LIN {X 0,Y 518.239,Z 318.605,A -85,B 0,C 180,E1 -4964.129,E2 -4964.129} C_VEL
LIN {X 0,Y 518.643,Z 306.673,A -85,B 0,C 180,E1 -4964.92,E2 -4964.92} C_VEL
LIN {X 0,Y 519.008,Z 293.496,A -85,B 0,C 180,E1 -4965.613,E2 -4965.613} C_VEL
LIN {X 0,Y 519.32,Z 279.565,A -85,B 0,C 180,E1 -4966.165,E2 -4966.165} C_VEL
LIN {X 0,Y 519.404,Z 270.973,A -85,B 0,C 180,E1 -4966.425,E2 -4966.425} C_VEL
LIN {X 0,Y 516.398,Z 257.452,A -85,B 0,C 180,E1 -4966.836,E2 -4966.836} C_VEL
LIN {X 0,Y 516.463,Z 251.755,A -85,B 0,C 180,E1 -4970.124,E2 -4970.124} C_VEL
LIN {X 0,Y 516.525,Z 246.395,A -85,B 0,C 180,E1 -4973.24,E2 -4973.24} C_VEL
LIN {X 0,Y 516.572,Z 241.654,A -85,B 0,C 180,E1 -4976.112,E2 -4976.112} C_VEL
LIN {X 0,Y 516.692,Z 236.476,A -85,B 0,C 180,E1 -4979.319,E2 -4979.319} C_VEL
LIN {X 0,Y 516.772,Z 231.444,A -85,B 0,C 180,E1 -4982.521,E2 -4982.521} C_VEL
LIN {X 0,Y 516.881,Z 227.139,A -85,B 0,C 180,E1 -4985.332,E2 -4985.332} C_VEL
LIN {X 0,Y 516.903,Z 223.246,A -85,B 0,C 180,E1 -4987.946,E2 -4987.946} C_VEL
LIN {X 0,Y 516.84,Z 221.733,A -85,B 0,C 180,E1 -4989.187,E2 -4989.187} C_VEL
LIN {X 0,Y 516.914,Z 221.722,A -85,B 0,C 180,E1 -4991.775,E2 -4991.775} C_VEL
LIN {X 0,Y 516.926,Z 221.721,A -85,B 0,C 180,E1 -4995.01,E2 -4995.01} C_VEL
LIN {X 0,Y 516.895,Z 221.723,A -85,B 0,C 180,E1 -4998.402,E2 -4998.402} C_VEL
LIN {X 0,Y 516.879,Z 221.728,A -85,B 0,C 180,E1 -5001.284,E2 -5001.284} C_VEL
LIN {X 0,Y 516.874,Z 221.728,A -85,B 0,C 180,E1 -5004.22,E2 -5004.22} C_VEL
LIN {X 0,Y 516.884,Z 221.723,A -85,B 0,C 180,E1 -5007.052,E2 -5007.052} C_VEL
LIN {X 0,Y 516.872,Z 221.725,A -85,B 0,C 180,E1 -5009.795,E2 -5009.795} C_VEL
LIN {X 0,Y 516.927,Z 221.723,A -85,B 0,C 180,E1 -5012.467,E2 -5012.467} C_VEL
LIN {X 0,Y 516.879,Z 221.722,A -85,B 0,C 180,E1 -5015.07,E2 -5015.07} C_VEL
LIN {X 0,Y 516.872,Z 221.727,A -85,B 0,C 180,E1 -5017.622,E2 -5017.622} C_VEL
LIN {X 0,Y 516.933,Z 221.717,A -85,B 0,C 180,E1 -5020.13,E2 -5020.13} C_VEL
LIN {X 0,Y 516.901,Z 221.723,A -85,B 0,C 180,E1 -5022.595,E2 -5022.595} C_VEL
LIN {X 0,Y 516.946,Z 221.716,A -85,B 0,C 180,E1 -5025.03,E2 -5025.03} C_VEL
LIN {X 0,Y 516.97,Z 221.713,A -85,B 0,C 180,E1 -5028.234,E2 -5028.234} C_VEL
LIN {X 0,Y 516.959,Z 221.714,A -85,B 0,C 180,E1 -5031.399,E2 -5031.399} C_VEL
LIN {X 0,Y 517.007,Z 221.711,A -85,B 0,C 180,E1 -5033.757,E2 -5033.757} C_VEL
LIN {X 0,Y 516.984,Z 221.715,A -85,B 0,C 180,E1 -5036.883,E2 -5036.883} C_VEL
LIN {X 0,Y 516.963,Z 221.719,A -85,B 0,C 180,E1 -5038.442,E2 -5038.442} C_VEL
LIN {X 0,Y 517.095,Z 221.697,A -85,B 0,C 180,E1 -5040.779,E2 -5040.779} C_VEL
LIN {X 0,Y 517.015,Z 221.71,A -85,B 0,C 180,E1 -5043.117,E2 -5043.117} C_VEL
LIN {X 0,Y 516.977,Z 221.714,A -85,B 0,C 180,E1 -5046.244,E2 -5046.244} C_VEL
LIN {X 0,Y 516.941,Z 221.718,A -85,B 0,C 180,E1 -5049.389,E2 -5049.389} C_VEL
LIN {X 0,Y 516.956,Z 221.715,A -85,B 0,C 180,E1 -5051.807,E2 -5051.807} C_VEL
LIN {X 0,Y 516.951,Z 221.716,A -85,B 0,C 180,E1 -5055.147,E2 -5055.147} C_VEL
LIN {X 0,Y 516.88,Z 221.725,A -85,B 0,C 180,E1 -5058.224,E2 -5058.224} C_VEL
LIN {X 0,Y 516.916,Z 221.721,A -85,B 0,C 180,E1 -5060.701,E2 -5060.701} C_VEL
LIN {X 0,Y 516.894,Z 221.724,A -85,B 0,C 180,E1 -5064.073,E2 -5064.073} C_VEL
LIN {X 0,Y 516.857,Z 221.726,A -85,B 0,C 180,E1 -5066.662,E2 -5066.662} C_VEL
LIN {X 0,Y 516.889,Z 221.725,A -85,B 0,C 180,E1 -5069.519,E2 -5069.519} C_VEL
LIN {X 0,Y 516.901,Z 221.726,A -85,B 0,C 180,E1 -5072.544,E2 -5072.544} C_VEL
LIN {X 0,Y 516.865,Z 221.728,A -85,B 0,C 180,E1 -5075.329,E2 -5075.329} C_VEL
LIN {X 0,Y 516.88,Z 221.725,A -85,B 0,C 180,E1 -5077.942,E2 -5077.942} C_VEL
LIN {X 0,Y 516.886,Z 221.728,A -85,B 0,C 180,E1 -5080.741,E2 -5080.741} C_VEL
LIN {X 0,Y 516.885,Z 221.726,A -85,B 0,C 180,E1 -5082.831,E2 -5082.831} C_VEL
LIN {X 0,Y 516.897,Z 221.726,A -85,B 0,C 180,E1 -5085.007,E2 -5085.007} C_VEL
LIN {X 0,Y 516.904,Z 221.724,A -85,B 0,C 180,E1 -5088.4,E2 -5088.4} C_VEL
LIN {X 0,Y 516.922,Z 221.812,A -85,B 0,C 180,E1 -5089.456,E2 -5089.456} C_VEL
LIN {X 0,Y 517.349,Z 225.366,A -85,B 0,C 180,E1 -5091.325,E2 -5091.325} C_VEL
LIN {X 0,Y 517.367,Z 229.331,A -85,B 0,C 180,E1 -5093.294,E2 -5093.294} C_VEL
LIN {X 0,Y 517.243,Z 235.304,A -85,B 0,C 180,E1 -5096.145,E2 -5096.145} C_VEL
LIN {X 0,Y 517.107,Z 241.306,A -85,B 0,C 180,E1 -5098.905,E2 -5098.905} C_VEL
LIN {X 0,Y 516.937,Z 248.486,A -85,B 0,C 180,E1 -5102.093,E2 -5102.093} C_VEL
LIN {X 0,Y 516.744,Z 255.392,A -85,B 0,C 180,E1 -5105.063,E2 -5105.063} C_VEL
LIN {X 0,Y 516.655,Z 261.572,A -85,B 0,C 180,E1 -5107.668,E2 -5107.668} C_VEL
LIN {X 0,Y 516.539,Z 268.467,A -85,B 0,C 180,E1 -5110.528,E2 -5110.528} C_VEL
LIN {X 0,Y 516.442,Z 275.13,A -85,B 0,C 180,E1 -5113.21,E2 -5113.21} C_VEL
LIN {X 0,Y 519.432,Z 289.702,A -85,B 0,C 180,E1 -5113.615,E2 -5113.615} C_VEL
LIN {X 0,Y 519.214,Z 303.013,A -85,B 0,C 180,E1 -5114.04,E2 -5114.04} C_VEL
LIN {X 0,Y 518.813,Z 315.653,A -85,B 0,C 180,E1 -5114.583,E2 -5114.583} C_VEL
LIN {X 0,Y 518.418,Z 328.162,A -85,B 0,C 180,E1 -5115.274,E2 -5115.274} C_VEL
LIN {X 0,Y 517.991,Z 340.984,A -85,B 0,C 180,E1 -5116.165,E2 -5116.165} C_VEL
LIN {X 0,Y 517.652,Z 352.544,A -85,B 0,C 180,E1 -5117.155,E2 -5117.155} C_VEL
LIN {X 0,Y 517.316,Z 363.018,A -85,B 0,C 180,E1 -5118.242,E2 -5118.242} C_VEL
LIN {X 0,Y 516.992,Z 372.482,A -85,B 0,C 180,E1 -5119.425,E2 -5119.425} C_VEL
LIN {X 0,Y 516.699,Z 381.498,A -85,B 0,C 180,E1 -5120.803,E2 -5120.803} C_VEL
LIN {X 0,Y 516.495,Z 388.781,A -85,B 0,C 180,E1 -5122.179,E2 -5122.179} C_VEL
LIN {X 0,Y 516.396,Z 395.328,A -85,B 0,C 180,E1 -5123.749,E2 -5123.749} C_VEL
LIN {X 0,Y 516.305,Z 399.157,A -85,B 0,C 180,E1 -5124.924,E2 -5124.924} C_VEL
LIN {X 0,Y 516.325,Z 402.109,A -85,B 0,C 180,E1 -5126.097,E2 -5126.097} C_VEL
LIN {X 0,Y 516.259,Z 404.809,A -85,B 0,C 180,E1 -5127.659,E2 -5127.659} C_VEL
LIN {X 0,Y 516.155,Z 406.146,A -85,B 0,C 180,E1 -5129.22,E2 -5129.22} C_VEL
LIN {X 0,Y 516.155,Z 406.147,A -85,B 0,C 180,E1 -5130.78,E2 -5130.78} C_VEL
LIN {X 0,Y 516.259,Z 404.812,A -85,B 0,C 180,E1 -5132.341,E2 -5132.341} C_VEL
LIN {X 0,Y 516.325,Z 402.113,A -85,B 0,C 180,E1 -5133.902,E2 -5133.902} C_VEL
LIN {X 0,Y 516.365,Z 397.974,A -85,B 0,C 180,E1 -5135.467,E2 -5135.467} C_VEL
LIN {X 0,Y 516.402,Z 392.27,A -85,B 0,C 180,E1 -5137.036,E2 -5137.036} C_VEL
LIN {X 0,Y 516.582,Z 385.842,A -85,B 0,C 180,E1 -5138.41,E2 -5138.41} C_VEL
LIN {X 0,Y 516.806,Z 377.856,A -85,B 0,C 180,E1 -5139.787,E2 -5139.787} C_VEL
LIN {X 0,Y 517.097,Z 369.503,A -85,B 0,C 180,E1 -5140.969,E2 -5140.969} C_VEL
LIN {X 0,Y 517.447,Z 359.048,A -85,B 0,C 180,E1 -5142.197,E2 -5142.197} C_VEL
LIN {X 0,Y 517.809,Z 348.231,A -85,B 0,C 180,E1 -5143.24,E2 -5143.24} C_VEL
LIN {X 0,Y 518.186,Z 335.647,A -85,B 0,C 180,E1 -5144.23,E2 -5144.23} C_VEL
LIN {X 0,Y 518.631,Z 323.158,A -85,B 0,C 180,E1 -5145.02,E2 -5145.02} C_VEL
LIN {X 0,Y 519.056,Z 310.322,A -85,B 0,C 180,E1 -5145.661,E2 -5145.661} C_VEL
LIN {X 0,Y 519.313,Z 296.904,A -85,B 0,C 180,E1 -5146.173,E2 -5146.173} C_VEL
LIN {X 0,Y 519.3,Z 289.202,A -85,B 0,C 180,E1 -5146.402,E2 -5146.402} C_VEL
LIN {X 0,Y 516.429,Z 274.971,A -85,B 0,C 180,E1 -5146.809,E2 -5146.809} C_VEL
LIN {X 0,Y 516.571,Z 266.806,A -85,B 0,C 180,E1 -5150.157,E2 -5150.157} C_VEL
LIN {X 0,Y 516.65,Z 259.421,A -85,B 0,C 180,E1 -5153.234,E2 -5153.234} C_VEL
LIN {X 0,Y 516.827,Z 252.503,A -85,B 0,C 180,E1 -5156.17,E2 -5156.17} C_VEL
LIN {X 0,Y 516.949,Z 246.322,A -85,B 0,C 180,E1 -5158.857,E2 -5158.857} C_VEL
LIN {X 0,Y 517.093,Z 241.291,A -85,B 0,C 180,E1 -5161.101,E2 -5161.101} C_VEL
LIN {X 0,Y 517.263,Z 234.923,A -85,B 0,C 180,E1 -5164.024,E2 -5164.024} C_VEL
LIN {X 0,Y 517.369,Z 229.265,A -85,B 0,C 180,E1 -5166.73,E2 -5166.73} C_VEL
LIN {X 0,Y 517.34,Z 225.355,A -85,B 0,C 180,E1 -5168.675,E2 -5168.675} C_VEL
LIN {X 0,Y 516.9,Z 221.726,A -85,B 0,C 180,E1 -5170.643,E2 -5170.643} C_VEL
LIN {X 0,Y 516.881,Z 221.726,A -85,B 0,C 180,E1 -5173.893,E2 -5173.893} C_VEL
LIN {X 0,Y 516.883,Z 221.73,A -85,B 0,C 180,E1 -5176.107,E2 -5176.107} C_VEL
LIN {X 0,Y 516.917,Z 221.72,A -85,B 0,C 180,E1 -5178.399,E2 -5178.399} C_VEL
LIN {X 0,Y 516.88,Z 221.728,A -85,B 0,C 180,E1 -5181.284,E2 -5181.284} C_VEL
LIN {X 0,Y 516.867,Z 221.731,A -85,B 0,C 180,E1 -5184.219,E2 -5184.219} C_VEL
LIN {X 0,Y 516.898,Z 221.723,A -85,B 0,C 180,E1 -5187.053,E2 -5187.053} C_VEL
LIN {X 0,Y 516.888,Z 221.723,A -85,B 0,C 180,E1 -5189.796,E2 -5189.796} C_VEL
LIN {X 0,Y 516.878,Z 221.729,A -85,B 0,C 180,E1 -5192.465,E2 -5192.465} C_VEL
LIN {X 0,Y 516.863,Z 221.726,A -85,B 0,C 180,E1 -5195.069,E2 -5195.069} C_VEL
LIN {X 0,Y 516.871,Z 221.727,A -85,B 0,C 180,E1 -5197.622,E2 -5197.622} C_VEL
LIN {X 0,Y 516.931,Z 221.719,A -85,B 0,C 180,E1 -5200.13,E2 -5200.13} C_VEL
LIN {X 0,Y 516.885,Z 221.724,A -85,B 0,C 180,E1 -5203.409,E2 -5203.409} C_VEL
LIN {X 0,Y 516.908,Z 221.72,A -85,B 0,C 180,E1 -5205.834,E2 -5205.834} C_VEL
LIN {X 0,Y 516.953,Z 221.714,A -85,B 0,C 180,E1 -5209.028,E2 -5209.028} C_VEL
LIN {X 0,Y 516.925,Z 221.72,A -85,B 0,C 180,E1 -5212.186,E2 -5212.186} C_VEL
LIN {X 0,Y 517.015,Z 221.707,A -85,B 0,C 180,E1 -5214.54,E2 -5214.54} C_VEL
LIN {X 0,Y 517.086,Z 221.698,A -85,B 0,C 180,E1 -5217.663,E2 -5217.663} C_VEL
LIN {X 0,Y 517.087,Z 221.703,A -85,B 0,C 180,E1 -5220,E2 -5220} C_VEL
LIN {X 0,Y 517.075,Z 221.699,A -85,B 0,C 180,E1 -5222.337,E2 -5222.337} C_VEL
LIN {X 0,Y 517.029,Z 221.705,A -85,B 0,C 180,E1 -5225.46,E2 -5225.46} C_VEL
LIN {X 0,Y 516.981,Z 221.713,A -85,B 0,C 180,E1 -5227.813,E2 -5227.813} C_VEL
LIN {X 0,Y 516.952,Z 221.716,A -85,B 0,C 180,E1 -5230.972,E2 -5230.972} C_VEL
LIN {X 0,Y 516.884,Z 221.724,A -85,B 0,C 180,E1 -5234.167,E2 -5234.167} C_VEL
LIN {X 0,Y 516.916,Z 221.721,A -85,B 0,C 180,E1 -5236.59,E2 -5236.59} C_VEL
LIN {X 0,Y 516.903,Z 221.722,A -85,B 0,C 180,E1 -5239.045,E2 -5239.045} C_VEL
LIN {X 0,Y 516.887,Z 221.723,A -85,B 0,C 180,E1 -5241.538,E2 -5241.538} C_VEL
LIN {X 0,Y 516.888,Z 221.728,A -85,B 0,C 180,E1 -5244.358,E2 -5244.358} C_VEL
LIN {X 0,Y 516.924,Z 221.718,A -85,B 0,C 180,E1 -5246.658,E2 -5246.658} C_VEL
LIN {X 0,Y 516.911,Z 221.721,A -85,B 0,C 180,E1 -5249.523,E2 -5249.523} C_VEL
LIN {X 0,Y 516.896,Z 221.726,A -85,B 0,C 180,E1 -5252.543,E2 -5252.543} C_VEL
LIN {X 0,Y 516.868,Z 221.727,A -85,B 0,C 180,E1 -5255.33,E2 -5255.33} C_VEL
LIN {X 0,Y 516.881,Z 221.723,A -85,B 0,C 180,E1 -5257.943,E2 -5257.943} C_VEL
LIN {X 0,Y 516.854,Z 221.731,A -85,B 0,C 180,E1 -5260.745,E2 -5260.745} C_VEL
LIN {X 0,Y 516.859,Z 221.727,A -85,B 0,C 180,E1 -5262.834,E2 -5262.834} C_VEL
LIN {X 0,Y 516.897,Z 221.724,A -85,B 0,C 180,E1 -5265.007,E2 -5265.007} C_VEL
LIN {X 0,Y 516.915,Z 221.724,A -85,B 0,C 180,E1 -5268.399,E2 -5268.399} C_VEL
LIN {X 0,Y 516.854,Z 221.732,A -85,B 0,C 180,E1 -5270.303,E2 -5270.303} C_VEL
LIN {X 0,Y 516.195,Z 222.043,A -85,B 0,C 180,E1 -5270.952,E2 -5270.952} C_VEL
LIN {X 0,Y 513.388,Z 223.496,A -85,B 0,C 180,E1 -5271.997,E2 -5271.997} C_VEL
LIN {X 0,Y 511,Z 225.03,A -85,B 0,C 180,E1 -5272.835,E2 -5272.835} C_VEL
LIN {X 0,Y 509.956,Z 226.113,A -85,B 0,C 180,E1 -5273.482,E2 -5273.482} C_VEL
LIN {X 0,Y 509.862,Z 226.448,A -85,B 0,C 180,E1 -5273.701,E2 -5273.701} C_VEL
LIN {X 0,Y 509.761,Z 230.691,A -85,B 0,C 180,E1 -5276.532,E2 -5276.532} C_VEL
LIN {X 0,Y 509.626,Z 234.981,A -85,B 0,C 180,E1 -5279.32,E2 -5279.32} C_VEL
LIN {X 0,Y 509.552,Z 239.246,A -85,B 0,C 180,E1 -5282.034,E2 -5282.034} C_VEL
LIN {X 0,Y 509.491,Z 243.501,A -85,B 0,C 180,E1 -5284.683,E2 -5284.683} C_VEL
LIN {X 0,Y 509.431,Z 248.25,A -85,B 0,C 180,E1 -5287.566,E2 -5287.566} C_VEL
LIN {X 0,Y 509.328,Z 253.534,A -85,B 0,C 180,E1 -5290.66,E2 -5290.66} C_VEL
LIN {X 0,Y 509.342,Z 257.614,A -85,B 0,C 180,E1 -5293.027,E2 -5293.027} C_VEL
LIN {X 0,Y 512.717,Z 272.931,A -85,B 0,C 180,E1 -5293.496,E2 -5293.496} C_VEL
LIN {X 0,Y 512.449,Z 285.258,A -85,B 0,C 180,E1 -5293.911,E2 -5293.911} C_VEL
LIN {X 0,Y 512.053,Z 297.91,A -85,B 0,C 180,E1 -5294.476,E2 -5294.476} C_VEL
LIN {X 0,Y 511.658,Z 310.151,A -85,B 0,C 180,E1 -5295.177,E2 -5295.177} C_VEL
LIN {X 0,Y 511.212,Z 322.746,A -85,B 0,C 180,E1 -5296.079,E2 -5296.079} C_VEL
LIN {X 0,Y 510.744,Z 334.116,A -85,B 0,C 180,E1 -5297.079,E2 -5297.079} C_VEL
LIN {X 0,Y 510.326,Z 343.538,A -85,B 0,C 180,E1 -5298.078,E2 -5298.078} C_VEL
LIN {X 0,Y 510.019,Z 352.998,A -85,B 0,C 180,E1 -5299.279,E2 -5299.279} C_VEL
LIN {X 0,Y 509.715,Z 362.026,A -85,B 0,C 180,E1 -5300.676,E2 -5300.676} C_VEL
LIN {X 0,Y 509.485,Z 369.293,A -85,B 0,C 180,E1 -5302.071,E2 -5302.071} C_VEL
LIN {X 0,Y 509.322,Z 375.819,A -85,B 0,C 180,E1 -5303.662,E2 -5303.662} C_VEL
LIN {X 0,Y 509.24,Z 379.655,A -85,B 0,C 180,E1 -5304.853,E2 -5304.853} C_VEL
LIN {X 0,Y 509.251,Z 382.596,A -85,B 0,C 180,E1 -5306.043,E2 -5306.043} C_VEL
LIN {X 0,Y 509.188,Z 385.306,A -85,B 0,C 180,E1 -5307.627,E2 -5307.627} C_VEL
LIN {X 0,Y 509.07,Z 386.669,A -85,B 0,C 180,E1 -5309.209,E2 -5309.209} C_VEL
LIN {X 0,Y 509.071,Z 386.711,A -85,B 0,C 180,E1 -5310.791,E2 -5310.791} C_VEL
LIN {X 0,Y 509.187,Z 385.428,A -85,B 0,C 180,E1 -5312.373,E2 -5312.373} C_VEL
LIN {X 0,Y 509.251,Z 382.793,A -85,B 0,C 180,E1 -5313.957,E2 -5313.957} C_VEL
LIN {X 0,Y 509.321,Z 378.738,A -85,B 0,C 180,E1 -5315.543,E2 -5315.543} C_VEL
LIN {X 0,Y 509.376,Z 373.135,A -85,B 0,C 180,E1 -5317.133,E2 -5317.133} C_VEL
LIN {X 0,Y 509.563,Z 366.806,A -85,B 0,C 180,E1 -5318.527,E2 -5318.527} C_VEL
LIN {X 0,Y 509.799,Z 358.936,A -85,B 0,C 180,E1 -5319.923,E2 -5319.923} C_VEL
LIN {X 0,Y 510.131,Z 350.7,A -85,B 0,C 180,E1 -5321.121,E2 -5321.121} C_VEL
LIN {X 0,Y 510.498,Z 341.042,A -85,B 0,C 180,E1 -5322.291,E2 -5322.291} C_VEL
LIN {X 0,Y 510.916,Z 329.731,A -85,B 0,C 180,E1 -5323.422,E2 -5323.422} C_VEL
LIN {X 0,Y 511.338,Z 318.732,A -85,B 0,C 180,E1 -5324.324,E2 -5324.324} C_VEL
LIN {X 0,Y 511.767,Z 306.797,A -85,B 0,C 180,E1 -5325.125,E2 -5325.125} C_VEL
LIN {X 0,Y 512.175,Z 293.617,A -85,B 0,C 180,E1 -5325.826,E2 -5325.826} C_VEL
LIN {X 0,Y 512.513,Z 279.691,A -85,B 0,C 180,E1 -5326.386,E2 -5326.386} C_VEL
LIN {X 0,Y 512.547,Z 272.007,A -85,B 0,C 180,E1 -5326.626,E2 -5326.626} C_VEL
LIN {X 0,Y 509.336,Z 257.59,A -85,B 0,C 180,E1 -5327.077,E2 -5327.077} C_VEL
LIN {X 0,Y 509.392,Z 252.115,A -85,B 0,C 180,E1 -5330.25,E2 -5330.25} C_VEL
LIN {X 0,Y 509.462,Z 246.484,A -85,B 0,C 180,E1 -5333.582,E2 -5333.582} C_VEL
LIN {X 0,Y 509.504,Z 242.087,A -85,B 0,C 180,E1 -5336.285,E2 -5336.285} C_VEL
LIN {X 0,Y 509.59,Z 237.976,A -85,B 0,C 180,E1 -5338.862,E2 -5338.862} C_VEL
LIN {X 0,Y 509.665,Z 233.699,A -85,B 0,C 180,E1 -5341.601,E2 -5341.601} C_VEL
LIN {X 0,Y 509.822,Z 229.401,A -85,B 0,C 180,E1 -5344.416,E2 -5344.416} C_VEL
LIN {X 0,Y 509.852,Z 225.073,A -85,B 0,C 180,E1 -5347.338,E2 -5347.338} C_VEL
LIN {X 0,Y 509.845,Z 223.63,A -85,B 0,C 180,E1 -5348.339,E2 -5348.339} C_VEL
LIN {X 0,Y 509.793,Z 222.612,A -85,B 0,C 180,E1 -5349.465,E2 -5349.465} C_VEL
LIN {X 0,Y 509.835,Z 222.602,A -85,B 0,C 180,E1 -5352.49,E2 -5352.49} C_VEL
LIN {X 0,Y 509.86,Z 222.599,A -85,B 0,C 180,E1 -5355.332,E2 -5355.332} C_VEL
LIN {X 0,Y 509.837,Z 222.602,A -85,B 0,C 180,E1 -5358.572,E2 -5358.572} C_VEL
LIN {X 0,Y 509.852,Z 222.599,A -85,B 0,C 180,E1 -5361.787,E2 -5361.787} C_VEL
LIN {X 0,Y 509.833,Z 222.605,A -85,B 0,C 180,E1 -5364.622,E2 -5364.622} C_VEL
LIN {X 0,Y 509.863,Z 222.602,A -85,B 0,C 180,E1 -5367.481,E2 -5367.481} C_VEL
LIN {X 0,Y 509.858,Z 222.599,A -85,B 0,C 180,E1 -5370.275,E2 -5370.275} C_VEL
LIN {X 0,Y 509.885,Z 222.596,A -85,B 0,C 180,E1 -5372.944,E2 -5372.944} C_VEL
LIN {X 0,Y 509.854,Z 222.601,A -85,B 0,C 180,E1 -5375.573,E2 -5375.573} C_VEL
LIN {X 0,Y 509.824,Z 222.602,A -85,B 0,C 180,E1 -5378.149,E2 -5378.149} C_VEL
LIN {X 0,Y 509.861,Z 222.603,A -85,B 0,C 180,E1 -5380.681,E2 -5380.681} C_VEL
LIN {X 0,Y 509.872,Z 222.597,A -85,B 0,C 180,E1 -5383.174,E2 -5383.174} C_VEL
LIN {X 0,Y 509.863,Z 222.601,A -85,B 0,C 180,E1 -5385.634,E2 -5385.634} C_VEL
LIN {X 0,Y 509.915,Z 222.594,A -85,B 0,C 180,E1 -5388.874,E2 -5388.874} C_VEL
LIN {X 0,Y 509.925,Z 222.594,A -85,B 0,C 180,E1 -5392.078,E2 -5392.078} C_VEL
LIN {X 0,Y 509.982,Z 222.582,A -85,B 0,C 180,E1 -5394.464,E2 -5394.464} C_VEL
LIN {X 0,Y 510.047,Z 222.574,A -85,B 0,C 180,E1 -5397.631,E2 -5397.631} C_VEL
LIN {X 0,Y 510.066,Z 222.572,A -85,B 0,C 180,E1 -5400.789,E2 -5400.789} C_VEL
LIN {X 0,Y 509.957,Z 222.589,A -85,B 0,C 180,E1 -5403.16,E2 -5403.16} C_VEL
LIN {X 0,Y 509.924,Z 222.593,A -85,B 0,C 180,E1 -5406.33,E2 -5406.33} C_VEL
LIN {X 0,Y 509.882,Z 222.598,A -85,B 0,C 180,E1 -5409.521,E2 -5409.521} C_VEL
LIN {X 0,Y 509.908,Z 222.592,A -85,B 0,C 180,E1 -5411.932,E2 -5411.932} C_VEL
LIN {X 0,Y 509.898,Z 222.594,A -85,B 0,C 180,E1 -5415.242,E2 -5415.242} C_VEL
LIN {X 0,Y 509.84,Z 222.601,A -85,B 0,C 180,E1 -5418.484,E2 -5418.484} C_VEL
LIN {X 0,Y 509.853,Z 222.603,A -85,B 0,C 180,E1 -5421.002,E2 -5421.002} C_VEL
LIN {X 0,Y 509.826,Z 222.602,A -85,B 0,C 180,E1 -5423.564,E2 -5423.564} C_VEL
LIN {X 0,Y 509.847,Z 222.601,A -85,B 0,C 180,E1 -5426.363,E2 -5426.363} C_VEL
LIN {X 0,Y 509.839,Z 222.602,A -85,B 0,C 180,E1 -5428.847,E2 -5428.847} C_VEL
LIN {X 0,Y 509.823,Z 222.602,A -85,B 0,C 180,E1 -5431.59,E2 -5431.59} C_VEL
LIN {X 0,Y 509.848,Z 222.603,A -85,B 0,C 180,E1 -5434.414,E2 -5434.414} C_VEL
LIN {X 0,Y 509.809,Z 222.611,A -85,B 0,C 180,E1 -5437.341,E2 -5437.341} C_VEL
LIN {X 0,Y 509.841,Z 222.605,A -85,B 0,C 180,E1 -5440.382,E2 -5440.382} C_VEL
LIN {X 0,Y 509.825,Z 222.605,A -85,B 0,C 180,E1 -5443.062,E2 -5443.062} C_VEL
LIN {X 0,Y 509.823,Z 222.607,A -85,B 0,C 180,E1 -5445.793,E2 -5445.793} C_VEL
LIN {X 0,Y 509.854,Z 222.607,A -85,B 0,C 180,E1 -5449.217,E2 -5449.217} C_VEL
LIN {X 0,Y 510.288,Z 225.328,A -85,B 0,C 180,E1 -5450.688,E2 -5450.688} C_VEL
LIN {X 0,Y 510.375,Z 229.88,A -85,B 0,C 180,E1 -5453.004,E2 -5453.004} C_VEL
LIN {X 0,Y 510.234,Z 235.493,A -85,B 0,C 180,E1 -5455.735,E2 -5455.735} C_VEL
LIN {X 0,Y 510.091,Z 241.771,A -85,B 0,C 180,E1 -5458.675,E2 -5458.675} C_VEL
LIN {X 0,Y 509.91,Z 248.906,A -85,B 0,C 180,E1 -5461.897,E2 -5461.897} C_VEL
LIN {X 0,Y 509.717,Z 255.305,A -85,B 0,C 180,E1 -5464.695,E2 -5464.695} C_VEL
LIN {X 0,Y 509.584,Z 261.896,A -85,B 0,C 180,E1 -5467.524,E2 -5467.524} C_VEL
LIN {X 0,Y 509.475,Z 268.324,A -85,B 0,C 180,E1 -5470.247,E2 -5470.247} C_VEL
LIN {X 0,Y 509.357,Z 274.989,A -85,B 0,C 180,E1 -5472.969,E2 -5472.969} C_VEL
LIN {X 0,Y 512.197,Z 288.849,A -85,B 0,C 180,E1 -5473.357,E2 -5473.357} C_VEL
LIN {X 0,Y 512.629,Z 292.205,A -85,B 0,C 180,E1 -5473.465,E2 -5473.465} C_VEL
LIN {X 0,Y 512.345,Z 305.416,A -85,B 0,C 180,E1 -5473.92,E2 -5473.92} C_VEL
LIN {X 0,Y 511.887,Z 317.508,A -85,B 0,C 180,E1 -5474.471,E2 -5474.471} C_VEL
LIN {X 0,Y 511.473,Z 329.611,A -85,B 0,C 180,E1 -5475.172,E2 -5475.172} C_VEL
LIN {X 0,Y 511.017,Z 342.143,A -85,B 0,C 180,E1 -5476.073,E2 -5476.073} C_VEL
LIN {X 0,Y 510.64,Z 353.477,A -85,B 0,C 180,E1 -5477.076,E2 -5477.076} C_VEL
LIN {X 0,Y 510.307,Z 362.882,A -85,B 0,C 180,E1 -5478.078,E2 -5478.078} C_VEL
LIN {X 0,Y 509.969,Z 372.347,A -85,B 0,C 180,E1 -5479.278,E2 -5479.278} C_VEL
LIN {X 0,Y 509.66,Z 381.363,A -85,B 0,C 180,E1 -5480.675,E2 -5480.675} C_VEL
LIN {X 0,Y 509.441,Z 388.646,A -85,B 0,C 180,E1 -5482.07,E2 -5482.07} C_VEL
LIN {X 0,Y 509.309,Z 395.192,A -85,B 0,C 180,E1 -5483.662,E2 -5483.662} C_VEL
LIN {X 0,Y 509.235,Z 399.022,A -85,B 0,C 180,E1 -5484.853,E2 -5484.853} C_VEL
LIN {X 0,Y 509.217,Z 401.973,A -85,B 0,C 180,E1 -5486.043,E2 -5486.043} C_VEL
LIN {X 0,Y 509.159,Z 404.674,A -85,B 0,C 180,E1 -5487.627,E2 -5487.627} C_VEL
LIN {X 0,Y 509.069,Z 406.012,A -85,B 0,C 180,E1 -5489.209,E2 -5489.209} C_VEL
LIN {X 0,Y 509.069,Z 406.012,A -85,B 0,C 180,E1 -5490.791,E2 -5490.791} C_VEL
LIN {X 0,Y 509.159,Z 404.678,A -85,B 0,C 180,E1 -5492.373,E2 -5492.373} C_VEL
LIN {X 0,Y 509.217,Z 401.978,A -85,B 0,C 180,E1 -5493.957,E2 -5493.957} C_VEL
LIN {X 0,Y 509.282,Z 397.839,A -85,B 0,C 180,E1 -5495.543,E2 -5495.543} C_VEL
LIN {X 0,Y 509.327,Z 392.135,A -85,B 0,C 180,E1 -5497.134,E2 -5497.134} C_VEL
LIN {X 0,Y 509.524,Z 385.707,A -85,B 0,C 180,E1 -5498.527,E2 -5498.527} C_VEL
LIN {X 0,Y 509.742,Z 377.72,A -85,B 0,C 180,E1 -5499.924,E2 -5499.924} C_VEL
LIN {X 0,Y 510.079,Z 369.367,A -85,B 0,C 180,E1 -5501.122,E2 -5501.122} C_VEL
LIN {X 0,Y 510.44,Z 359.266,A -85,B 0,C 180,E1 -5502.327,E2 -5502.327} C_VEL
LIN {X 0,Y 510.836,Z 348.095,A -85,B 0,C 180,E1 -5503.424,E2 -5503.424} C_VEL
LIN {X 0,Y 511.207,Z 336.939,A -85,B 0,C 180,E1 -5504.327,E2 -5504.327} C_VEL
LIN {X 0,Y 511.656,Z 324.793,A -85,B 0,C 180,E1 -5505.128,E2 -5505.128} C_VEL
LIN {X 0,Y 512.183,Z 311.319,A -85,B 0,C 180,E1 -5505.826,E2 -5505.826} C_VEL
LIN {X 0,Y 512.478,Z 297.439,A -85,B 0,C 180,E1 -5506.372,E2 -5506.372} C_VEL
LIN {X 0,Y 512.534,Z 290.629,A -85,B 0,C 180,E1 -5506.581,E2 -5506.581} C_VEL
LIN {X 0,Y 509.419,Z 275.626,A -85,B 0,C 180,E1 -5507.018,E2 -5507.018} C_VEL
LIN {X 0,Y 509.333,Z 274.83,A -85,B 0,C 180,E1 -5507.051,E2 -5507.051} C_VEL
LIN {X 0,Y 509.511,Z 267.047,A -85,B 0,C 180,E1 -5510.287,E2 -5510.287} C_VEL
LIN {X 0,Y 509.588,Z 260.343,A -85,B 0,C 180,E1 -5513.145,E2 -5513.145} C_VEL
LIN {X 0,Y 509.78,Z 253.285,A -85,B 0,C 180,E1 -5516.178,E2 -5516.178} C_VEL
LIN {X 0,Y 509.916,Z 247.249,A -85,B 0,C 180,E1 -5518.842,E2 -5518.842} C_VEL
LIN {X 0,Y 510.067,Z 241.231,A -85,B 0,C 180,E1 -5521.573,E2 -5521.573} C_VEL
LIN {X 0,Y 510.239,Z 235.229,A -85,B 0,C 180,E1 -5524.384,E2 -5524.384} C_VEL
LIN {X 0,Y 510.382,Z 229.268,A -85,B 0,C 180,E1 -5527.293,E2 -5527.293} C_VEL
LIN {X 0,Y 510.201,Z 224.929,A -85,B 0,C 180,E1 -5529.52,E2 -5529.52} C_VEL
LIN {X 0,Y 509.863,Z 222.603,A -85,B 0,C 180,E1 -5530.831,E2 -5530.831} C_VEL
LIN {X 0,Y 509.822,Z 222.606,A -85,B 0,C 180,E1 -5534.207,E2 -5534.207} C_VEL
LIN {X 0,Y 509.824,Z 222.604,A -85,B 0,C 180,E1 -5536.938,E2 -5536.938} C_VEL
LIN {X 0,Y 509.84,Z 222.605,A -85,B 0,C 180,E1 -5539.618,E2 -5539.618} C_VEL
LIN {X 0,Y 509.808,Z 222.611,A -85,B 0,C 180,E1 -5542.658,E2 -5542.658} C_VEL
LIN {X 0,Y 509.856,Z 222.604,A -85,B 0,C 180,E1 -5545.798,E2 -5545.798} C_VEL
LIN {X 0,Y 509.847,Z 222.601,A -85,B 0,C 180,E1 -5548.72,E2 -5548.72} C_VEL
LIN {X 0,Y 509.849,Z 222.601,A -85,B 0,C 180,E1 -5551.154,E2 -5551.154} C_VEL
LIN {X 0,Y 509.866,Z 222.6,A -85,B 0,C 180,E1 -5553.827,E2 -5553.827} C_VEL
LIN {X 0,Y 509.824,Z 222.603,A -85,B 0,C 180,E1 -5556.436,E2 -5556.436} C_VEL
LIN {X 0,Y 509.918,Z 222.591,A -85,B 0,C 180,E1 -5559.845,E2 -5559.845} C_VEL
LIN {X 0,Y 509.854,Z 222.598,A -85,B 0,C 180,E1 -5563.174,E2 -5563.174} C_VEL
LIN {X 0,Y 509.876,Z 222.598,A -85,B 0,C 180,E1 -5565.634,E2 -5565.634} C_VEL
LIN {X 0,Y 509.915,Z 222.592,A -85,B 0,C 180,E1 -5568.875,E2 -5568.875} C_VEL
LIN {X 0,Y 509.878,Z 222.599,A -85,B 0,C 180,E1 -5572.077,E2 -5572.077} C_VEL
LIN {X 0,Y 509.966,Z 222.585,A -85,B 0,C 180,E1 -5574.464,E2 -5574.464} C_VEL
LIN {X 0,Y 510.057,Z 222.573,A -85,B 0,C 180,E1 -5577.631,E2 -5577.631} C_VEL
LIN {X 0,Y 510.058,Z 222.579,A -85,B 0,C 180,E1 -5580,E2 -5580} C_VEL
LIN {X 0,Y 510.046,Z 222.574,A -85,B 0,C 180,E1 -5582.369,E2 -5582.369} C_VEL
LIN {X 0,Y 509.98,Z 222.583,A -85,B 0,C 180,E1 -5585.536,E2 -5585.536} C_VEL
LIN {X 0,Y 509.954,Z 222.59,A -85,B 0,C 180,E1 -5587.922,E2 -5587.922} C_VEL
LIN {X 0,Y 509.914,Z 222.594,A -85,B 0,C 180,E1 -5591.126,E2 -5591.126} C_VEL
LIN {X 0,Y 509.856,Z 222.601,A -85,B 0,C 180,E1 -5594.366,E2 -5594.366} C_VEL
LIN {X 0,Y 509.885,Z 222.595,A -85,B 0,C 180,E1 -5596.825,E2 -5596.825} C_VEL
LIN {X 0,Y 509.918,Z 222.59,A -85,B 0,C 180,E1 -5600.155,E2 -5600.155} C_VEL
LIN {X 0,Y 509.823,Z 222.602,A -85,B 0,C 180,E1 -5603.564,E2 -5603.564} C_VEL
LIN {X 0,Y 509.912,Z 222.592,A -85,B 0,C 180,E1 -5606.378,E2 -5606.378} C_VEL
LIN {X 0,Y 509.874,Z 222.598,A -85,B 0,C 180,E1 -5608.845,E2 -5608.845} C_VEL
LIN {X 0,Y 509.82,Z 222.603,A -85,B 0,C 180,E1 -5611.59,E2 -5611.59} C_VEL
LIN {X 0,Y 509.841,Z 222.602,A -85,B 0,C 180,E1 -5614.414,E2 -5614.414} C_VEL
LIN {X 0,Y 509.818,Z 222.609,A -85,B 0,C 180,E1 -5617.341,E2 -5617.341} C_VEL
LIN {X 0,Y 509.815,Z 222.607,A -85,B 0,C 180,E1 -5620.385,E2 -5620.385} C_VEL
LIN {X 0,Y 509.805,Z 222.606,A -85,B 0,C 180,E1 -5623.06,E2 -5623.06} C_VEL
LIN {X 0,Y 509.824,Z 222.605,A -85,B 0,C 180,E1 -5625.793,E2 -5625.793} C_VEL
LIN {X 0,Y 509.856,Z 222.605,A -85,B 0,C 180,E1 -5628.574,E2 -5628.574} C_VEL
LIN {X 0,Y 509.824,Z 222.608,A -85,B 0,C 180,E1 -5630.645,E2 -5630.645} C_VEL
LIN {X 0,Y 509.864,Z 223.661,A -85,B 0,C 180,E1 -5631.785,E2 -5631.785} C_VEL
LIN {X 0,Y 509.862,Z 226.448,A -85,B 0,C 180,E1 -5633.701,E2 -5633.701} C_VEL
LIN {X 0,Y 509.167,Z 227.502,A -85,B 0,C 180,E1 -5634.35,E2 -5634.35} C_VEL
LIN {X 0,Y 506.289,Z 229.425,A -85,B 0,C 180,E1 -5635.399,E2 -5635.399} C_VEL
LIN {X 0,Y 503.854,Z 230.986,A -85,B 0,C 180,E1 -5636.243,E2 -5636.243} C_VEL
LIN {X 0,Y 502.786,Z 232.094,A -85,B 0,C 180,E1 -5636.897,E2 -5636.897} C_VEL
LIN {X 0,Y 502.687,Z 232.439,A -85,B 0,C 180,E1 -5637.119,E2 -5637.119} C_VEL
LIN {X 0,Y 502.562,Z 237.015,A -85,B 0,C 180,E1 -5640.116,E2 -5640.116} C_VEL
LIN {X 0,Y 502.457,Z 240.756,A -85,B 0,C 180,E1 -5642.511,E2 -5642.511} C_VEL
LIN {X 0,Y 502.439,Z 245.345,A -85,B 0,C 180,E1 -5645.396,E2 -5645.396} C_VEL
LIN {X 0,Y 502.357,Z 249.307,A -85,B 0,C 180,E1 -5647.807,E2 -5647.807} C_VEL
LIN {X 0,Y 502.278,Z 253.634,A -85,B 0,C 180,E1 -5650.378,E2 -5650.378} C_VEL
LIN {X 0,Y 502.268,Z 257.732,A -85,B 0,C 180,E1 -5652.781,E2 -5652.781} C_VEL
LIN {X 0,Y 505.763,Z 273.081,A -85,B 0,C 180,E1 -5653.262,E2 -5653.262} C_VEL
LIN {X 0,Y 505.626,Z 285.409,A -85,B 0,C 180,E1 -5653.688,E2 -5653.688} C_VEL
LIN {X 0,Y 505.233,Z 298.057,A -85,B 0,C 180,E1 -5654.261,E2 -5654.261} C_VEL
LIN {X 0,Y 504.805,Z 310.296,A -85,B 0,C 180,E1 -5654.971,E2 -5654.971} C_VEL
LIN {X 0,Y 504.321,Z 322.889,A -85,B 0,C 180,E1 -5655.885,E2 -5655.885} C_VEL
LIN {X 0,Y 503.805,Z 334.257,A -85,B 0,C 180,E1 -5656.898,E2 -5656.898} C_VEL
LIN {X 0,Y 503.322,Z 345.394,A -85,B 0,C 180,E1 -5658.114,E2 -5658.114} C_VEL
LIN {X 0,Y 502.956,Z 354.542,A -85,B 0,C 180,E1 -5659.33,E2 -5659.33} C_VEL
LIN {X 0,Y 502.629,Z 363.276,A -85,B 0,C 180,E1 -5660.747,E2 -5660.747} C_VEL
LIN {X 0,Y 502.443,Z 369.431,A -85,B 0,C 180,E1 -5661.959,E2 -5661.959} C_VEL
LIN {X 0,Y 502.255,Z 375.956,A -85,B 0,C 180,E1 -5663.573,E2 -5663.573} C_VEL
LIN {X 0,Y 502.177,Z 379.791,A -85,B 0,C 180,E1 -5664.781,E2 -5664.781} C_VEL
LIN {X 0,Y 502.148,Z 382.733,A -85,B 0,C 180,E1 -5665.987,E2 -5665.987} C_VEL
LIN {X 0,Y 502.09,Z 385.441,A -85,B 0,C 180,E1 -5667.593,E2 -5667.593} C_VEL
LIN {X 0,Y 501.987,Z 386.803,A -85,B 0,C 180,E1 -5669.198,E2 -5669.198} C_VEL
LIN {X 0,Y 501.988,Z 386.845,A -85,B 0,C 180,E1 -5670.802,E2 -5670.802} C_VEL
LIN {X 0,Y 502.089,Z 385.562,A -85,B 0,C 180,E1 -5672.407,E2 -5672.407} C_VEL
LIN {X 0,Y 502.148,Z 382.927,A -85,B 0,C 180,E1 -5674.013,E2 -5674.013} C_VEL
LIN {X 0,Y 502.256,Z 378.871,A -85,B 0,C 180,E1 -5675.621,E2 -5675.621} C_VEL
LIN {X 0,Y 502.318,Z 373.268,A -85,B 0,C 180,E1 -5677.234,E2 -5677.234} C_VEL
LIN {X 0,Y 502.531,Z 366.938,A -85,B 0,C 180,E1 -5678.647,E2 -5678.647} C_VEL
LIN {X 0,Y 502.773,Z 359.067,A -85,B 0,C 180,E1 -5680.063,E2 -5680.063} C_VEL
LIN {X 0,Y 503.136,Z 350.831,A -85,B 0,C 180,E1 -5681.277,E2 -5681.277} C_VEL
LIN {X 0,Y 503.548,Z 340.91,A -85,B 0,C 180,E1 -5682.493,E2 -5682.493} C_VEL
LIN {X 0,Y 503.995,Z 329.859,A -85,B 0,C 180,E1 -5683.61,E2 -5683.61} C_VEL
LIN {X 0,Y 504.446,Z 318.859,A -85,B 0,C 180,E1 -5684.524,E2 -5684.524} C_VEL
LIN {X 0,Y 504.906,Z 306.922,A -85,B 0,C 180,E1 -5685.336,E2 -5685.336} C_VEL
LIN {X 0,Y 505.354,Z 293.737,A -85,B 0,C 180,E1 -5686.046,E2 -5686.046} C_VEL
LIN {X 0,Y 505.714,Z 279.638,A -85,B 0,C 180,E1 -5686.618,E2 -5686.618} C_VEL
LIN {X 0,Y 505.712,Z 273.134,A -85,B 0,C 180,E1 -5686.828,E2 -5686.828} C_VEL
LIN {X 0,Y 502.677,Z 259.782,A -85,B 0,C 180,E1 -5687.254,E2 -5687.254} C_VEL
LIN {X 0,Y 502.28,Z 257.717,A -85,B 0,C 180,E1 -5687.318,E2 -5687.318} C_VEL
LIN {X 0,Y 502.321,Z 252.34,A -85,B 0,C 180,E1 -5690.474,E2 -5690.474} C_VEL
LIN {X 0,Y 502.373,Z 248.01,A -85,B 0,C 180,E1 -5693.061,E2 -5693.061} C_VEL
LIN {X 0,Y 502.419,Z 243.745,A -85,B 0,C 180,E1 -5695.699,E2 -5695.699} C_VEL
LIN {X 0,Y 502.512,Z 239.483,A -85,B 0,C 180,E1 -5698.393,E2 -5698.393} C_VEL
LIN {X 0,Y 502.606,Z 234.735,A -85,B 0,C 180,E1 -5701.463,E2 -5701.463} C_VEL
LIN {X 0,Y 502.776,Z 230.248,A -85,B 0,C 180,E1 -5704.439,E2 -5704.439} C_VEL
LIN {X 0,Y 502.812,Z 226.242,A -85,B 0,C 180,E1 -5707.183,E2 -5707.183} C_VEL
LIN {X 0,Y 502.74,Z 223.68,A -85,B 0,C 180,E1 -5708.982,E2 -5708.982} C_VEL
LIN {X 0,Y 502.801,Z 223.483,A -85,B 0,C 180,E1 -5711.068,E2 -5711.068} C_VEL
LIN {X 0,Y 502.793,Z 223.482,A -85,B 0,C 180,E1 -5714.339,E2 -5714.339} C_VEL
LIN {X 0,Y 502.76,Z 223.485,A -85,B 0,C 180,E1 -5716.767,E2 -5716.767} C_VEL
LIN {X 0,Y 502.773,Z 223.482,A -85,B 0,C 180,E1 -5719.012,E2 -5719.012} C_VEL
LIN {X 0,Y 502.795,Z 223.478,A -85,B 0,C 180,E1 -5722.046,E2 -5722.046} C_VEL
LIN {X 0,Y 502.799,Z 223.478,A -85,B 0,C 180,E1 -5725.034,E2 -5725.034} C_VEL
LIN {X 0,Y 502.785,Z 223.482,A -85,B 0,C 180,E1 -5727.915,E2 -5727.915} C_VEL
LIN {X 0,Y 502.823,Z 223.478,A -85,B 0,C 180,E1 -5730.712,E2 -5730.712} C_VEL
LIN {X 0,Y 502.866,Z 223.469,A -85,B 0,C 180,E1 -5733.439,E2 -5733.439} C_VEL
LIN {X 0,Y 502.779,Z 223.482,A -85,B 0,C 180,E1 -5736.085,E2 -5736.085} C_VEL
LIN {X 0,Y 502.784,Z 223.482,A -85,B 0,C 180,E1 -5738.689,E2 -5738.689} C_VEL
LIN {X 0,Y 502.826,Z 223.474,A -85,B 0,C 180,E1 -5741.248,E2 -5741.248} C_VEL
LIN {X 0,Y 502.852,Z 223.47,A -85,B 0,C 180,E1 -5744.6,E2 -5744.6} C_VEL
LIN {X 0,Y 502.88,Z 223.467,A -85,B 0,C 180,E1 -5748.039,E2 -5748.039} C_VEL
LIN {X 0,Y 502.867,Z 223.469,A -85,B 0,C 180,E1 -5751.157,E2 -5751.157} C_VEL
LIN {X 0,Y 502.911,Z 223.469,A -85,B 0,C 180,E1 -5753.581,E2 -5753.581} C_VEL
LIN {X 0,Y 502.873,Z 223.473,A -85,B 0,C 180,E1 -5756.795,E2 -5756.795} C_VEL
LIN {X 0,Y 502.901,Z 223.47,A -85,B 0,C 180,E1 -5758.398,E2 -5758.398} C_VEL
LIN {X 0,Y 503.036,Z 223.448,A -85,B 0,C 180,E1 -5760.8,E2 -5760.8} C_VEL
LIN {X 0,Y 502.9,Z 223.469,A -85,B 0,C 180,E1 -5763.204,E2 -5763.204} C_VEL
LIN {X 0,Y 502.874,Z 223.472,A -85,B 0,C 180,E1 -5766.419,E2 -5766.419} C_VEL
LIN {X 0,Y 502.831,Z 223.478,A -85,B 0,C 180,E1 -5769.655,E2 -5769.655} C_VEL
LIN {X 0,Y 502.85,Z 223.471,A -85,B 0,C 180,E1 -5772.102,E2 -5772.102} C_VEL
LIN {X 0,Y 502.851,Z 223.471,A -85,B 0,C 180,E1 -5775.4,E2 -5775.4} C_VEL
LIN {X 0,Y 502.814,Z 223.476,A -85,B 0,C 180,E1 -5778.752,E2 -5778.752} C_VEL
LIN {X 0,Y 502.786,Z 223.483,A -85,B 0,C 180,E1 -5781.311,E2 -5781.311} C_VEL
LIN {X 0,Y 502.777,Z 223.481,A -85,B 0,C 180,E1 -5783.914,E2 -5783.914} C_VEL
LIN {X 0,Y 502.791,Z 223.479,A -85,B 0,C 180,E1 -5786.57,E2 -5786.57} C_VEL
LIN {X 0,Y 502.812,Z 223.476,A -85,B 0,C 180,E1 -5789.934,E2 -5789.934} C_VEL
LIN {X 0,Y 502.835,Z 223.474,A -85,B 0,C 180,E1 -5793.031,E2 -5793.031} C_VEL
LIN {X 0,Y 502.769,Z 223.486,A -85,B 0,C 180,E1 -5795.952,E2 -5795.952} C_VEL
LIN {X 0,Y 502.803,Z 223.483,A -85,B 0,C 180,E1 -5798.976,E2 -5798.976} C_VEL
LIN {X 0,Y 502.799,Z 223.484,A -85,B 0,C 180,E1 -5802.139,E2 -5802.139} C_VEL
LIN {X 0,Y 502.787,Z 223.485,A -85,B 0,C 180,E1 -5805.47,E2 -5805.47} C_VEL
LIN {X 0,Y 502.85,Z 223.517,A -85,B 0,C 180,E1 -5809.039,E2 -5809.039} C_VEL
LIN {X 0,Y 503.364,Z 227.948,A -85,B 0,C 180,E1 -5811.433,E2 -5811.433} C_VEL
LIN {X 0,Y 503.368,Z 231.215,A -85,B 0,C 180,E1 -5813.104,E2 -5813.104} C_VEL
LIN {X 0,Y 503.198,Z 237.179,A -85,B 0,C 180,E1 -5816.036,E2 -5816.036} C_VEL
LIN {X 0,Y 503.033,Z 243.167,A -85,B 0,C 180,E1 -5818.873,E2 -5818.873} C_VEL
LIN {X 0,Y 502.883,Z 249.335,A -85,B 0,C 180,E1 -5821.697,E2 -5821.697} C_VEL
LIN {X 0,Y 502.662,Z 256.224,A -85,B 0,C 180,E1 -5824.758,E2 -5824.758} C_VEL
LIN {X 0,Y 502.515,Z 263.232,A -85,B 0,C 180,E1 -5827.814,E2 -5827.814} C_VEL
LIN {X 0,Y 502.397,Z 269.195,A -85,B 0,C 180,E1 -5830.383,E2 -5830.383} C_VEL
LIN {X 0,Y 502.28,Z 274.849,A -85,B 0,C 180,E1 -5832.722,E2 -5832.722} C_VEL
LIN {X 0,Y 505.275,Z 289.495,A -85,B 0,C 180,E1 -5833.145,E2 -5833.145} C_VEL
LIN {X 0,Y 505.802,Z 293.371,A -85,B 0,C 180,E1 -5833.273,E2 -5833.273} C_VEL
LIN {X 0,Y 505.458,Z 307.393,A -85,B 0,C 180,E1 -5833.784,E2 -5833.784} C_VEL
LIN {X 0,Y 504.977,Z 319.339,A -85,B 0,C 180,E1 -5834.356,E2 -5834.356} C_VEL
LIN {X 0,Y 504.489,Z 332.514,A -85,B 0,C 180,E1 -5835.168,E2 -5835.168} C_VEL
LIN {X 0,Y 504.021,Z 344.43,A -85,B 0,C 180,E1 -5836.082,E2 -5836.082} C_VEL
LIN {X 0,Y 503.514,Z 356.391,A -85,B 0,C 180,E1 -5837.208,E2 -5837.208} C_VEL
LIN {X 0,Y 503.164,Z 366.072,A -85,B 0,C 180,E1 -5838.315,E2 -5838.315} C_VEL
LIN {X 0,Y 502.821,Z 374.955,A -85,B 0,C 180,E1 -5839.531,E2 -5839.531} C_VEL
LIN {X 0,Y 502.519,Z 383.467,A -85,B 0,C 180,E1 -5840.948,E2 -5840.948} C_VEL
LIN {X 0,Y 502.318,Z 390.328,A -85,B 0,C 180,E1 -5842.362,E2 -5842.362} C_VEL
LIN {X 0,Y 502.234,Z 395.057,A -85,B 0,C 180,E1 -5843.572,E2 -5843.572} C_VEL
LIN {X 0,Y 502.103,Z 399.956,A -85,B 0,C 180,E1 -5845.182,E2 -5845.182} C_VEL
LIN {X 0,Y 502.112,Z 403.363,A -85,B 0,C 180,E1 -5846.79,E2 -5846.79} C_VEL
LIN {X 0,Y 502.032,Z 405.377,A -85,B 0,C 180,E1 -5848.396,E2 -5848.396} C_VEL
LIN {X 0,Y 501.978,Z 406.044,A -85,B 0,C 180,E1 -5850,E2 -5850} C_VEL
LIN {X 0,Y 502.032,Z 405.379,A -85,B 0,C 180,E1 -5851.604,E2 -5851.604} C_VEL
LIN {X 0,Y 502.112,Z 403.367,A -85,B 0,C 180,E1 -5853.209,E2 -5853.209} C_VEL
LIN {X 0,Y 502.103,Z 399.959,A -85,B 0,C 180,E1 -5854.817,E2 -5854.817} C_VEL
LIN {X 0,Y 502.234,Z 395.056,A -85,B 0,C 180,E1 -5856.428,E2 -5856.428} C_VEL
LIN {X 0,Y 502.37,Z 388.511,A -85,B 0,C 180,E1 -5858.042,E2 -5858.042} C_VEL
LIN {X 0,Y 502.614,Z 381.229,A -85,B 0,C 180,E1 -5859.456,E2 -5859.456} C_VEL
LIN {X 0,Y 502.944,Z 372.212,A -85,B 0,C 180,E1 -5860.874,E2 -5860.874} C_VEL
LIN {X 0,Y 503.302,Z 362.748,A -85,B 0,C 180,E1 -5862.09,E2 -5862.09} C_VEL
LIN {X 0,Y 503.694,Z 352.273,A -85,B 0,C 180,E1 -5863.207,E2 -5863.207} C_VEL
LIN {X 0,Y 504.142,Z 340.716,A -85,B 0,C 180,E1 -5864.223,E2 -5864.223} C_VEL
LIN {X 0,Y 504.666,Z 327.898,A -85,B 0,C 180,E1 -5865.136,E2 -5865.136} C_VEL
LIN {X 0,Y 505.154,Z 315.381,A -85,B 0,C 180,E1 -5865.845,E2 -5865.845} C_VEL
LIN {X 0,Y 505.518,Z 301.994,A -85,B 0,C 180,E1 -5866.434,E2 -5866.434} C_VEL
LIN {X 0,Y 505.643,Z 291.428,A -85,B 0,C 180,E1 -5866.788,E2 -5866.788} C_VEL
LIN {X 0,Y 502.569,Z 276.588,A -85,B 0,C 180,E1 -5867.238,E2 -5867.238} C_VEL
LIN {X 0,Y 502.281,Z 274.69,A -85,B 0,C 180,E1 -5867.297,E2 -5867.297} C_VEL
LIN {X 0,Y 502.432,Z 267.205,A -85,B 0,C 180,E1 -5870.469,E2 -5870.469} C_VEL
LIN {X 0,Y 502.562,Z 260.25,A -85,B 0,C 180,E1 -5873.488,E2 -5873.488} C_VEL
LIN {X 0,Y 502.755,Z 253.199,A -85,B 0,C 180,E1 -5876.572,E2 -5876.572} C_VEL
LIN {X 0,Y 502.899,Z 247.168,A -85,B 0,C 180,E1 -5879.283,E2 -5879.283} C_VEL
LIN {X 0,Y 503.103,Z 241.16,A -85,B 0,C 180,E1 -5882.062,E2 -5882.062} C_VEL
LIN {X 0,Y 503.231,Z 235.171,A -85,B 0,C 180,E1 -5884.932,E2 -5884.932} C_VEL
LIN {X 0,Y 503.374,Z 229.221,A -85,B 0,C 180,E1 -5887.903,E2 -5887.903} C_VEL
LIN {X 0,Y 503.094,Z 225.276,A -85,B 0,C 180,E1 -5889.986,E2 -5889.986} C_VEL
LIN {X 0,Y 502.831,Z 223.478,A -85,B 0,C 180,E1 -5891.065,E2 -5891.065} C_VEL
LIN {X 0,Y 502.786,Z 223.484,A -85,B 0,C 180,E1 -5894.53,E2 -5894.53} C_VEL
LIN {X 0,Y 502.798,Z 223.483,A -85,B 0,C 180,E1 -5897.861,E2 -5897.861} C_VEL
LIN {X 0,Y 502.802,Z 223.483,A -85,B 0,C 180,E1 -5901.024,E2 -5901.024} C_VEL
LIN {X 0,Y 502.771,Z 223.487,A -85,B 0,C 180,E1 -5904.17,E2 -5904.17} C_VEL
LIN {X 0,Y 502.834,Z 223.475,A -85,B 0,C 180,E1 -5906.993,E2 -5906.993} C_VEL
LIN {X 0,Y 502.815,Z 223.476,A -85,B 0,C 180,E1 -5910.065,E2 -5910.065} C_VEL
LIN {X 0,Y 502.8,Z 223.478,A -85,B 0,C 180,E1 -5913.454,E2 -5913.454} C_VEL
LIN {X 0,Y 502.775,Z 223.482,A -85,B 0,C 180,E1 -5916.085,E2 -5916.085} C_VEL
LIN {X 0,Y 502.785,Z 223.483,A -85,B 0,C 180,E1 -5918.689,E2 -5918.689} C_VEL
LIN {X 0,Y 502.812,Z 223.476,A -85,B 0,C 180,E1 -5921.248,E2 -5921.248} C_VEL
LIN {X 0,Y 502.839,Z 223.472,A -85,B 0,C 180,E1 -5924.664,E2 -5924.664} C_VEL
LIN {X 0,Y 502.879,Z 223.468,A -85,B 0,C 180,E1 -5928.039,E2 -5928.039} C_VEL
LIN {X 0,Y 502.852,Z 223.471,A -85,B 0,C 180,E1 -5931.156,E2 -5931.156} C_VEL
LIN {X 0,Y 502.919,Z 223.462,A -85,B 0,C 180,E1 -5934.386,E2 -5934.386} C_VEL
LIN {X 0,Y 503.027,Z 223.449,A -85,B 0,C 180,E1 -5937.598,E2 -5937.598} C_VEL
LIN {X 0,Y 503.029,Z 223.454,A -85,B 0,C 180,E1 -5940,E2 -5940} C_VEL
LIN {X 0,Y 503.015,Z 223.45,A -85,B 0,C 180,E1 -5942.402,E2 -5942.402} C_VEL
LIN {X 0,Y 502.934,Z 223.461,A -85,B 0,C 180,E1 -5945.614,E2 -5945.614} C_VEL
LIN {X 0,Y 502.904,Z 223.469,A -85,B 0,C 180,E1 -5948.033,E2 -5948.033} C_VEL
LIN {X 0,Y 502.879,Z 223.473,A -85,B 0,C 180,E1 -5951.283,E2 -5951.283} C_VEL
LIN {X 0,Y 502.841,Z 223.478,A -85,B 0,C 180,E1 -5954.571,E2 -5954.571} C_VEL
LIN {X 0,Y 502.858,Z 223.475,A -85,B 0,C 180,E1 -5957.907,E2 -5957.907} C_VEL
LIN {X 0,Y 502.831,Z 223.474,A -85,B 0,C 180,E1 -5960.536,E2 -5960.536} C_VEL
LIN {X 0,Y 502.789,Z 223.48,A -85,B 0,C 180,E1 -5963.041,E2 -5963.041} C_VEL
LIN {X 0,Y 502.823,Z 223.477,A -85,B 0,C 180,E1 -5965.677,E2 -5965.677} C_VEL
LIN {X 0,Y 502.839,Z 223.472,A -85,B 0,C 180,E1 -5968.373,E2 -5968.373} C_VEL
LIN {X 0,Y 502.794,Z 223.478,A -85,B 0,C 180,E1 -5971.499,E2 -5971.499} C_VEL
LIN {X 0,Y 502.792,Z 223.484,A -85,B 0,C 180,E1 -5973.995,E2 -5973.995} C_VEL
LIN {X 0,Y 502.779,Z 223.485,A -85,B 0,C 180,E1 -5977.178,E2 -5977.178} C_VEL
LIN {X 0,Y 502.772,Z 223.481,A -85,B 0,C 180,E1 -5980.017,E2 -5980.017} C_VEL
LIN {X 0,Y 502.776,Z 223.487,A -85,B 0,C 180,E1 -5982.196,E2 -5982.196} C_VEL
LIN {X 0,Y 502.788,Z 223.484,A -85,B 0,C 180,E1 -5985.47,E2 -5985.47} C_VEL
LIN {X 0,Y 502.797,Z 223.48,A -85,B 0,C 180,E1 -5987.861,E2 -5987.861} C_VEL
LIN {X 0,Y 502.754,Z 223.544,A -85,B 0,C 180,E1 -5991.019,E2 -5991.019} C_VEL
LIN {X 0,Y 502.807,Z 227.343,A -85,B 0,C 180,E1 -5993.681,E2 -5993.681} C_VEL
LIN {X 0,Y 502.745,Z 230.759,A -85,B 0,C 180,E1 -5996.002,E2 -5996.002} C_VEL
LIN {X 0,Y 502.687,Z 232.439,A -85,B 0,C 180,E1 -5997.119,E2 -5997.119} C_VEL
LIN {X 0,Y 501.982,Z 233.513,A -85,B 0,C 180,E1 -5997.776,E2 -5997.776} C_VEL
LIN {X 0,Y 499.09,Z 235.461,A -85,B 0,C 180,E1 -5998.839,E2 -5998.839} C_VEL
LIN {X 0,Y 496.646,Z 237.043,A -85,B 0,C 180,E1 -5999.694,E2 -5999.694} C_VEL
LIN {X 0,Y 495.572,Z 238.17,A -85,B 0,C 180,E1 -6000.357,E2 -6000.357} C_VEL
LIN {X 0,Y 495.471,Z 238.525,A -85,B 0,C 180,E1 -6000.582,E2 -6000.582} C_VEL
LIN {X 0,Y 495.36,Z 243.689,A -85,B 0,C 180,E1 -6003.908,E2 -6003.908} C_VEL
LIN {X 0,Y 495.302,Z 247.963,A -85,B 0,C 180,E1 -6006.59,E2 -6006.59} C_VEL
LIN {X 0,Y 495.245,Z 252.75,A -85,B 0,C 180,E1 -6009.489,E2 -6009.489} C_VEL
LIN {X 0,Y 495.206,Z 257.837,A -85,B 0,C 180,E1 -6012.521,E2 -6012.521} C_VEL
LIN {X 0,Y 498.846,Z 273.706,A -85,B 0,C 180,E1 -6013.037,E2 -6013.037} C_VEL
LIN {X 0,Y 499.024,Z 277.345,A -85,B 0,C 180,E1 -6013.16,E2 -6013.16} C_VEL
LIN {X 0,Y 498.692,Z 289.664,A -85,B 0,C 180,E1 -6013.629,E2 -6013.629} C_VEL
LIN {X 0,Y 498.273,Z 302.03,A -85,B 0,C 180,E1 -6014.246,E2 -6014.246} C_VEL
LIN {X 0,Y 497.731,Z 314.953,A -85,B 0,C 180,E1 -6015.067,E2 -6015.067} C_VEL
LIN {X 0,Y 497.224,Z 326.662,A -85,B 0,C 180,E1 -6015.992,E2 -6015.992} C_VEL
LIN {X 0,Y 496.724,Z 337.468,A -85,B 0,C 180,E1 -6017.03,E2 -6017.03} C_VEL
LIN {X 0,Y 496.299,Z 347.332,A -85,B 0,C 180,E1 -6018.174,E2 -6018.174} C_VEL
LIN {X 0,Y 495.874,Z 356.03,A -85,B 0,C 180,E1 -6019.383,E2 -6019.383} C_VEL
LIN {X 0,Y 495.557,Z 364.526,A -85,B 0,C 180,E1 -6020.819,E2 -6020.819} C_VEL
LIN {X 0,Y 495.322,Z 371.369,A -85,B 0,C 180,E1 -6022.253,E2 -6022.253} C_VEL
LIN {X 0,Y 495.173,Z 376.925,A -85,B 0,C 180,E1 -6023.721,E2 -6023.721} C_VEL
LIN {X 0,Y 495.033,Z 380.988,A -85,B 0,C 180,E1 -6025.114,E2 -6025.114} C_VEL
LIN {X 0,Y 495.038,Z 384.395,A -85,B 0,C 180,E1 -6026.745,E2 -6026.745} C_VEL
LIN {X 0,Y 494.961,Z 386.423,A -85,B 0,C 180,E1 -6028.373,E2 -6028.373} C_VEL
LIN {X 0,Y 494.897,Z 387.124,A -85,B 0,C 180,E1 -6030,E2 -6030} C_VEL
LIN {X 0,Y 494.959,Z 386.504,A -85,B 0,C 180,E1 -6031.627,E2 -6031.627} C_VEL
LIN {X 0,Y 495.038,Z 384.55,A -85,B 0,C 180,E1 -6033.256,E2 -6033.256} C_VEL
LIN {X 0,Y 495.032,Z 381.218,A -85,B 0,C 180,E1 -6034.887,E2 -6034.887} C_VEL
LIN {X 0,Y 495.165,Z 377.267,A -85,B 0,C 180,E1 -6036.271,E2 -6036.271} C_VEL
LIN {X 0,Y 495.316,Z 371.764,A -85,B 0,C 180,E1 -6037.747,E2 -6037.747} C_VEL
LIN {X 0,Y 495.55,Z 365.01,A -85,B 0,C 180,E1 -6039.181,E2 -6039.181} C_VEL
LIN {X 0,Y 495.844,Z 356.617,A -85,B 0,C 180,E1 -6040.618,E2 -6040.618} C_VEL
LIN {X 0,Y 496.318,Z 346.859,A -85,B 0,C 180,E1 -6041.976,E2 -6041.976} C_VEL
LIN {X 0,Y 496.729,Z 337.239,A -85,B 0,C 180,E1 -6043.084,E2 -6043.084} C_VEL
LIN {X 0,Y 497.243,Z 326.499,A -85,B 0,C 180,E1 -6044.112,E2 -6044.112} C_VEL
LIN {X 0,Y 497.754,Z 314.748,A -85,B 0,C 180,E1 -6045.037,E2 -6045.037} C_VEL
LIN {X 0,Y 498.224,Z 303.54,A -85,B 0,C 180,E1 -6045.756,E2 -6045.756} C_VEL
LIN {X 0,Y 498.678,Z 290.6,A -85,B 0,C 180,E1 -6046.418,E2 -6046.418} C_VEL
LIN {X 0,Y 499.005,Z 277.402,A -85,B 0,C 180,E1 -6046.929,E2 -6046.929} C_VEL
LIN {X 0,Y 498.849,Z 274.017,A -85,B 0,C 180,E1 -6047.045,E2 -6047.045} C_VEL
LIN {X 0,Y 495.824,Z 260.592,A -85,B 0,C 180,E1 -6047.488,E2 -6047.488} C_VEL
LIN {X 0,Y 495.214,Z 257.812,A -85,B 0,C 180,E1 -6047.583,E2 -6047.583} C_VEL
LIN {X 0,Y 495.231,Z 252.451,A -85,B 0,C 180,E1 -6050.78,E2 -6050.78} C_VEL
LIN {X 0,Y 495.304,Z 248.111,A -85,B 0,C 180,E1 -6053.41,E2 -6053.41} C_VEL
LIN {X 0,Y 495.361,Z 243.84,A -85,B 0,C 180,E1 -6056.092,E2 -6056.092} C_VEL
LIN {X 0,Y 495.452,Z 239.57,A -85,B 0,C 180,E1 -6058.835,E2 -6058.835} C_VEL
LIN {X 0,Y 495.574,Z 235.217,A -85,B 0,C 180,E1 -6061.691,E2 -6061.691} C_VEL
LIN {X 0,Y 495.755,Z 230.761,A -85,B 0,C 180,E1 -6064.691,E2 -6064.691} C_VEL
LIN {X 0,Y 495.777,Z 226.64,A -85,B 0,C 180,E1 -6067.558,E2 -6067.558} C_VEL
LIN {X 0,Y 495.733,Z 224.948,A -85,B 0,C 180,E1 -6068.763,E2 -6068.763} C_VEL
LIN {X 0,Y 495.725,Z 224.366,A -85,B 0,C 180,E1 -6070.042,E2 -6070.042} C_VEL
LIN {X 0,Y 495.728,Z 224.363,A -85,B 0,C 180,E1 -6072.883,E2 -6072.883} C_VEL
LIN {X 0,Y 495.733,Z 224.361,A -85,B 0,C 180,E1 -6075.999,E2 -6075.999} C_VEL
LIN {X 0,Y 495.733,Z 224.361,A -85,B 0,C 180,E1 -6079.297,E2 -6079.297} C_VEL
LIN {X 0,Y 495.748,Z 224.359,A -85,B 0,C 180,E1 -6081.408,E2 -6081.408} C_VEL
LIN {X 0,Y 495.75,Z 224.361,A -85,B 0,C 180,E1 -6084.462,E2 -6084.462} C_VEL
LIN {X 0,Y 495.769,Z 224.356,A -85,B 0,C 180,E1 -6087.406,E2 -6087.406} C_VEL
LIN {X 0,Y 495.765,Z 224.354,A -85,B 0,C 180,E1 -6090.253,E2 -6090.253} C_VEL
LIN {X 0,Y 495.827,Z 224.346,A -85,B 0,C 180,E1 -6093.251,E2 -6093.251} C_VEL
LIN {X 0,Y 495.746,Z 224.356,A -85,B 0,C 180,E1 -6096.613,E2 -6096.613} C_VEL
LIN {X 0,Y 495.782,Z 224.353,A -85,B 0,C 180,E1 -6099.324,E2 -6099.324} C_VEL
LIN {X 0,Y 495.782,Z 224.353,A -85,B 0,C 180,E1 -6101.828,E2 -6101.828} C_VEL
LIN {X 0,Y 495.828,Z 224.346,A -85,B 0,C 180,E1 -6104.548,E2 -6104.548} C_VEL
LIN {X 0,Y 495.832,Z 224.345,A -85,B 0,C 180,E1 -6107.965,E2 -6107.965} C_VEL
LIN {X 0,Y 495.837,Z 224.345,A -85,B 0,C 180,E1 -6111.03,E2 -6111.03} C_VEL
LIN {X 0,Y 495.865,Z 224.346,A -85,B 0,C 180,E1 -6113.489,E2 -6113.489} C_VEL
LIN {X 0,Y 495.819,Z 224.352,A -85,B 0,C 180,E1 -6116.75,E2 -6116.75} C_VEL
LIN {X 0,Y 495.871,Z 224.345,A -85,B 0,C 180,E1 -6118.376,E2 -6118.376} C_VEL
LIN {X 0,Y 495.986,Z 224.326,A -85,B 0,C 180,E1 -6120.812,E2 -6120.812} C_VEL
LIN {X 0,Y 495.996,Z 224.324,A -85,B 0,C 180,E1 -6122.436,E2 -6122.436} C_VEL
LIN {X 0,Y 495.875,Z 224.34,A -85,B 0,C 180,E1 -6125.694,E2 -6125.694} C_VEL
LIN {X 0,Y 495.811,Z 224.348,A -85,B 0,C 180,E1 -6128.97,E2 -6128.97} C_VEL
LIN {X 0,Y 495.832,Z 224.345,A -85,B 0,C 180,E1 -6132.035,E2 -6132.035} C_VEL
LIN {X 0,Y 495.826,Z 224.346,A -85,B 0,C 180,E1 -6135.451,E2 -6135.451} C_VEL
LIN {X 0,Y 495.774,Z 224.353,A -85,B 0,C 180,E1 -6139.029,E2 -6139.029} C_VEL
LIN {X 0,Y 495.746,Z 224.357,A -85,B 0,C 180,E1 -6141.629,E2 -6141.629} C_VEL
LIN {X 0,Y 495.724,Z 224.364,A -85,B 0,C 180,E1 -6144.276,E2 -6144.276} C_VEL
LIN {X 0,Y 495.736,Z 224.357,A -85,B 0,C 180,E1 -6146.979,E2 -6146.979} C_VEL
LIN {X 0,Y 495.761,Z 224.354,A -85,B 0,C 180,E1 -6150.146,E2 -6150.146} C_VEL
LIN {X 0,Y 495.795,Z 224.35,A -85,B 0,C 180,E1 -6153.244,E2 -6153.244} C_VEL
LIN {X 0,Y 495.713,Z 224.364,A -85,B 0,C 180,E1 -6156.087,E2 -6156.087} C_VEL
LIN {X 0,Y 495.764,Z 224.359,A -85,B 0,C 180,E1 -6158.768,E2 -6158.768} C_VEL
LIN {X 0,Y 495.759,Z 224.358,A -85,B 0,C 180,E1 -6161.781,E2 -6161.781} C_VEL
LIN {X 0,Y 495.739,Z 224.363,A -85,B 0,C 180,E1 -6165.141,E2 -6165.141} C_VEL
LIN {X 0,Y 495.801,Z 224.44,A -85,B 0,C 180,E1 -6168.859,E2 -6168.859} C_VEL
LIN {X 0,Y 496.373,Z 229.188,A -85,B 0,C 180,E1 -6171.465,E2 -6171.465} C_VEL
LIN {X 0,Y 496.276,Z 233.78,A -85,B 0,C 180,E1 -6173.824,E2 -6173.824} C_VEL
LIN {X 0,Y 496.13,Z 239.579,A -85,B 0,C 180,E1 -6176.697,E2 -6176.697} C_VEL
LIN {X 0,Y 495.934,Z 246.148,A -85,B 0,C 180,E1 -6179.82,E2 -6179.82} C_VEL
LIN {X 0,Y 495.743,Z 253.117,A -85,B 0,C 180,E1 -6183.021,E2 -6183.021} C_VEL
LIN {X 0,Y 495.527,Z 260.154,A -85,B 0,C 180,E1 -6186.158,E2 -6186.158} C_VEL
LIN {X 0,Y 495.377,Z 267.605,A -85,B 0,C 180,E1 -6189.448,E2 -6189.448} C_VEL
LIN {X 0,Y 495.208,Z 274.558,A -85,B 0,C 180,E1 -6192.447,E2 -6192.447} C_VEL
LIN {X 0,Y 498.691,Z 291.78,A -85,B 0,C 180,E1 -6192.985,E2 -6192.985} C_VEL
LIN {X 0,Y 498.951,Z 295.192,A -85,B 0,C 180,E1 -6193.102,E2 -6193.102} C_VEL
LIN {X 0,Y 498.573,Z 308.793,A -85,B 0,C 180,E1 -6193.625,E2 -6193.625} C_VEL
LIN {X 0,Y 498.052,Z 320.98,A -85,B 0,C 180,E1 -6194.238,E2 -6194.238} C_VEL
LIN {X 0,Y 497.536,Z 333.807,A -85,B 0,C 180,E1 -6195.061,E2 -6195.061} C_VEL
LIN {X 0,Y 497.049,Z 345.471,A -85,B 0,C 180,E1 -6195.987,E2 -6195.987} C_VEL
LIN {X 0,Y 496.557,Z 356.255,A -85,B 0,C 180,E1 -6197.026,E2 -6197.026} C_VEL
LIN {X 0,Y 496.144,Z 366.212,A -85,B 0,C 180,E1 -6198.182,E2 -6198.182} C_VEL
LIN {X 0,Y 495.801,Z 374.82,A -85,B 0,C 180,E1 -6199.381,E2 -6199.381} C_VEL
LIN {X 0,Y 495.471,Z 383.332,A -85,B 0,C 180,E1 -6200.818,E2 -6200.818} C_VEL
LIN {X 0,Y 495.235,Z 390.192,A -85,B 0,C 180,E1 -6202.252,E2 -6202.252} C_VEL
LIN {X 0,Y 495.121,Z 395.91,A -85,B 0,C 180,E1 -6203.762,E2 -6203.762} C_VEL
LIN {X 0,Y 495.03,Z 399.821,A -85,B 0,C 180,E1 -6205.113,E2 -6205.113} C_VEL
LIN {X 0,Y 495.033,Z 403.228,A -85,B 0,C 180,E1 -6206.744,E2 -6206.744} C_VEL
LIN {X 0,Y 494.958,Z 405.243,A -85,B 0,C 180,E1 -6208.373,E2 -6208.373} C_VEL
LIN {X 0,Y 494.896,Z 405.91,A -85,B 0,C 180,E1 -6210,E2 -6210} C_VEL
LIN {X 0,Y 494.958,Z 405.244,A -85,B 0,C 180,E1 -6211.627,E2 -6211.627} C_VEL
LIN {X 0,Y 495.033,Z 403.233,A -85,B 0,C 180,E1 -6213.255,E2 -6213.255} C_VEL
LIN {X 0,Y 495.03,Z 399.825,A -85,B 0,C 180,E1 -6214.886,E2 -6214.886} C_VEL
LIN {X 0,Y 495.131,Z 395.033,A -85,B 0,C 180,E1 -6216.488,E2 -6216.488} C_VEL
LIN {X 0,Y 495.235,Z 390.192,A -85,B 0,C 180,E1 -6217.748,E2 -6217.748} C_VEL
LIN {X 0,Y 495.47,Z 383.334,A -85,B 0,C 180,E1 -6219.182,E2 -6219.182} C_VEL
LIN {X 0,Y 495.801,Z 374.82,A -85,B 0,C 180,E1 -6220.619,E2 -6220.619} C_VEL
LIN {X 0,Y 496.193,Z 365.067,A -85,B 0,C 180,E1 -6221.962,E2 -6221.962} C_VEL
LIN {X 0,Y 496.603,Z 355.18,A -85,B 0,C 180,E1 -6223.087,E2 -6223.087} C_VEL
LIN {X 0,Y 497.075,Z 344.296,A -85,B 0,C 180,E1 -6224.116,E2 -6224.116} C_VEL
LIN {X 0,Y 497.575,Z 332.384,A -85,B 0,C 180,E1 -6225.043,E2 -6225.043} C_VEL
LIN {X 0,Y 498.141,Z 319.204,A -85,B 0,C 180,E1 -6225.864,E2 -6225.864} C_VEL
LIN {X 0,Y 498.615,Z 306.332,A -85,B 0,C 180,E1 -6226.486,E2 -6226.486} C_VEL
LIN {X 0,Y 498.822,Z 292.443,A -85,B 0,C 180,E1 -6226.991,E2 -6226.991} C_VEL
LIN {X 0,Y 495.871,Z 278.132,A -85,B 0,C 180,E1 -6227.448,E2 -6227.448} C_VEL
LIN {X 0,Y 495.208,Z 274.558,A -85,B 0,C 180,E1 -6227.553,E2 -6227.553} C_VEL
LIN {X 0,Y 495.376,Z 267.604,A -85,B 0,C 180,E1 -6230.552,E2 -6230.552} C_VEL
LIN {X 0,Y 495.5,Z 261.142,A -85,B 0,C 180,E1 -6233.4,E2 -6233.4} C_VEL
LIN {X 0,Y 495.724,Z 253.666,A -85,B 0,C 180,E1 -6236.726,E2 -6236.726} C_VEL
LIN {X 0,Y 495.883,Z 247.081,A -85,B 0,C 180,E1 -6239.739,E2 -6239.739} C_VEL
LIN {X 0,Y 496.098,Z 241.088,A -85,B 0,C 180,E1 -6242.57,E2 -6242.57} C_VEL
LIN {X 0,Y 496.239,Z 235.112,A -85,B 0,C 180,E1 -6245.497,E2 -6245.497} C_VEL
LIN {X 0,Y 496.371,Z 229.173,A -85,B 0,C 180,E1 -6248.535,E2 -6248.535} C_VEL
LIN {X 0,Y 495.801,Z 224.426,A -85,B 0,C 180,E1 -6251.141,E2 -6251.141} C_VEL
LIN {X 0,Y 495.724,Z 224.362,A -85,B 0,C 180,E1 -6254.002,E2 -6254.002} C_VEL
LIN {X 0,Y 495.726,Z 224.361,A -85,B 0,C 180,E1 -6257.117,E2 -6257.117} C_VEL
LIN {X 0,Y 495.76,Z 224.356,A -85,B 0,C 180,E1 -6259.953,E2 -6259.953} C_VEL
LIN {X 0,Y 495.719,Z 224.365,A -85,B 0,C 180,E1 -6262.555,E2 -6262.555} C_VEL
LIN {X 0,Y 495.777,Z 224.355,A -85,B 0,C 180,E1 -6265.457,E2 -6265.457} C_VEL
LIN {X 0,Y 495.757,Z 224.355,A -85,B 0,C 180,E1 -6268.364,E2 -6268.364} C_VEL
LIN {X 0,Y 495.734,Z 224.359,A -85,B 0,C 180,E1 -6271.183,E2 -6271.183} C_VEL
LIN {X 0,Y 495.738,Z 224.362,A -85,B 0,C 180,E1 -6273.929,E2 -6273.929} C_VEL
LIN {X 0,Y 495.761,Z 224.359,A -85,B 0,C 180,E1 -6277.14,E2 -6277.14} C_VEL
LIN {X 0,Y 495.769,Z 224.355,A -85,B 0,C 180,E1 -6280.11,E2 -6280.11} C_VEL
LIN {X 0,Y 495.744,Z 224.356,A -85,B 0,C 180,E1 -6282.68,E2 -6282.68} C_VEL
LIN {X 0,Y 495.796,Z 224.353,A -85,B 0,C 180,E1 -6285.217,E2 -6285.217} C_VEL
LIN {X 0,Y 495.854,Z 224.347,A -85,B 0,C 180,E1 -6288.555,E2 -6288.555} C_VEL
LIN {X 0,Y 495.815,Z 224.353,A -85,B 0,C 180,E1 -6291.851,E2 -6291.851} C_VEL
LIN {X 0,Y 495.874,Z 224.34,A -85,B 0,C 180,E1 -6294.306,E2 -6294.306} C_VEL
LIN {X 0,Y 495.995,Z 224.325,A -85,B 0,C 180,E1 -6297.564,E2 -6297.564} C_VEL
LIN {X 0,Y 496,Z 224.33,A -85,B 0,C 180,E1 -6300,E2 -6300} C_VEL
LIN {X 0,Y 495.984,Z 224.326,A -85,B 0,C 180,E1 -6302.436,E2 -6302.436} C_VEL
LIN {X 0,Y 495.891,Z 224.338,A -85,B 0,C 180,E1 -6305.694,E2 -6305.694} C_VEL
LIN {X 0,Y 495.875,Z 224.345,A -85,B 0,C 180,E1 -6308.148,E2 -6308.148} C_VEL
LIN {X 0,Y 495.853,Z 224.347,A -85,B 0,C 180,E1 -6311.445,E2 -6311.445} C_VEL
LIN {X 0,Y 495.788,Z 224.354,A -85,B 0,C 180,E1 -6314.783,E2 -6314.783} C_VEL
LIN {X 0,Y 495.784,Z 224.352,A -85,B 0,C 180,E1 -6317.319,E2 -6317.319} C_VEL
LIN {X 0,Y 495.772,Z 224.353,A -85,B 0,C 180,E1 -6319.89,E2 -6319.89} C_VEL
LIN {X 0,Y 495.76,Z 224.358,A -85,B 0,C 180,E1 -6322.86,E2 -6322.86} C_VEL
LIN {X 0,Y 495.783,Z 224.356,A -85,B 0,C 180,E1 -6326.068,E2 -6326.068} C_VEL
LIN {X 0,Y 495.771,Z 224.355,A -85,B 0,C 180,E1 -6328.815,E2 -6328.815} C_VEL
LIN {X 0,Y 495.756,Z 224.355,A -85,B 0,C 180,E1 -6331.725,E2 -6331.725} C_VEL
LIN {X 0,Y 495.765,Z 224.354,A -85,B 0,C 180,E1 -6334.693,E2 -6334.693} C_VEL
LIN {X 0,Y 495.731,Z 224.361,A -85,B 0,C 180,E1 -6337.562,E2 -6337.562} C_VEL
LIN {X 0,Y 495.745,Z 224.357,A -85,B 0,C 180,E1 -6340.045,E2 -6340.045} C_VEL
LIN {X 0,Y 495.71,Z 224.362,A -85,B 0,C 180,E1 -6342.885,E2 -6342.885} C_VEL
LIN {X 0,Y 495.73,Z 224.36,A -85,B 0,C 180,E1 -6345.998,E2 -6345.998} C_VEL
LIN {X 0,Y 495.741,Z 224.363,A -85,B 0,C 180,E1 -6348.709,E2 -6348.709} C_VEL
LIN {X 0,Y 495.738,Z 224.363,A -85,B 0,C 180,E1 -6350.36,E2 -6350.36} C_VEL
LIN {X 0,Y 495.751,Z 225.054,A -85,B 0,C 180,E1 -6351.408,E2 -6351.408} C_VEL
LIN {X 0,Y 495.762,Z 228.589,A -85,B 0,C 180,E1 -6353.905,E2 -6353.905} C_VEL
LIN {X 0,Y 495.685,Z 232.266,A -85,B 0,C 180,E1 -6356.43,E2 -6356.43} C_VEL
LIN {X 0,Y 495.524,Z 236.567,A -85,B 0,C 180,E1 -6359.297,E2 -6359.297} C_VEL
LIN {X 0,Y 495.471,Z 238.525,A -85,B 0,C 180,E1 -6360.582,E2 -6360.582} C_VEL
LIN {X 0,Y 494.758,Z 239.627,A -85,B 0,C 180,E1 -6361.248,E2 -6361.248} C_VEL
LIN {X 0,Y 491.855,Z 241.6,A -85,B 0,C 180,E1 -6362.325,E2 -6362.325} C_VEL
LIN {X 0,Y 489.42,Z 243.195,A -85,B 0,C 180,E1 -6363.193,E2 -6363.193} C_VEL
LIN {X 0,Y 488.372,Z 244.341,A -85,B 0,C 180,E1 -6363.865,E2 -6363.865} C_VEL
LIN {X 0,Y 488.284,Z 244.704,A -85,B 0,C 180,E1 -6364.093,E2 -6364.093} C_VEL
LIN {X 0,Y 488.254,Z 248.067,A -85,B 0,C 180,E1 -6366.232,E2 -6366.232} C_VEL
LIN {X 0,Y 488.165,Z 253.163,A -85,B 0,C 180,E1 -6369.357,E2 -6369.357} C_VEL
LIN {X 0,Y 488.122,Z 257.957,A -85,B 0,C 180,E1 -6372.252,E2 -6372.252} C_VEL
LIN {X 0,Y 491.857,Z 273.965,A -85,B 0,C 180,E1 -6372.791,E2 -6372.791} C_VEL
LIN {X 0,Y 492.237,Z 277.235,A -85,B 0,C 180,E1 -6372.911,E2 -6372.911} C_VEL
LIN {X 0,Y 491.85,Z 290.939,A -85,B 0,C 180,E1 -6373.448,E2 -6373.448} C_VEL
LIN {X 0,Y 491.392,Z 303.938,A -85,B 0,C 180,E1 -6374.126,E2 -6374.126} C_VEL
LIN {X 0,Y 490.804,Z 316.518,A -85,B 0,C 180,E1 -6374.957,E2 -6374.957} C_VEL
LIN {X 0,Y 490.264,Z 327.974,A -85,B 0,C 180,E1 -6375.895,E2 -6375.895} C_VEL
LIN {X 0,Y 489.729,Z 338.679,A -85,B 0,C 180,E1 -6376.958,E2 -6376.958} C_VEL
LIN {X 0,Y 489.259,Z 349.134,A -85,B 0,C 180,E1 -6378.217,E2 -6378.217} C_VEL
LIN {X 0,Y 488.756,Z 358.804,A -85,B 0,C 180,E1 -6379.645,E2 -6379.645} C_VEL
LIN {X 0,Y 488.456,Z 366.771,A -85,B 0,C 180,E1 -6381.102,E2 -6381.102} C_VEL
LIN {X 0,Y 488.187,Z 373.185,A -85,B 0,C 180,E1 -6382.556,E2 -6382.556} C_VEL
LIN {X 0,Y 488.116,Z 378.87,A -85,B 0,C 180,E1 -6384.216,E2 -6384.216} C_VEL
LIN {X 0,Y 487.949,Z 383.006,A -85,B 0,C 180,E1 -6385.87,E2 -6385.87} C_VEL
LIN {X 0,Y 487.907,Z 385.713,A -85,B 0,C 180,E1 -6387.523,E2 -6387.523} C_VEL
LIN {X 0,Y 487.831,Z 387.073,A -85,B 0,C 180,E1 -6389.175,E2 -6389.175} C_VEL
LIN {X 0,Y 487.832,Z 387.114,A -85,B 0,C 180,E1 -6390.826,E2 -6390.826} C_VEL
LIN {X 0,Y 487.906,Z 385.83,A -85,B 0,C 180,E1 -6392.477,E2 -6392.477} C_VEL
LIN {X 0,Y 487.949,Z 383.194,A -85,B 0,C 180,E1 -6394.13,E2 -6394.13} C_VEL
LIN {X 0,Y 488.103,Z 379.137,A -85,B 0,C 180,E1 -6395.785,E2 -6395.785} C_VEL
LIN {X 0,Y 488.185,Z 373.533,A -85,B 0,C 180,E1 -6397.445,E2 -6397.445} C_VEL
LIN {X 0,Y 488.447,Z 367.202,A -85,B 0,C 180,E1 -6398.898,E2 -6398.898} C_VEL
LIN {X 0,Y 488.721,Z 359.33,A -85,B 0,C 180,E1 -6400.356,E2 -6400.356} C_VEL
LIN {X 0,Y 489.184,Z 351.092,A -85,B 0,C 180,E1 -6401.603,E2 -6401.603} C_VEL
LIN {X 0,Y 489.622,Z 340.545,A -85,B 0,C 180,E1 -6402.929,E2 -6402.929} C_VEL
LIN {X 0,Y 490.187,Z 330.116,A -85,B 0,C 180,E1 -6404.001,E2 -6404.001} C_VEL
LIN {X 0,Y 490.685,Z 319.113,A -85,B 0,C 180,E1 -6404.94,E2 -6404.94} C_VEL
LIN {X 0,Y 491.212,Z 307.171,A -85,B 0,C 180,E1 -6405.774,E2 -6405.774} C_VEL
LIN {X 0,Y 491.737,Z 293.979,A -85,B 0,C 180,E1 -6406.503,E2 -6406.503} C_VEL
LIN {X 0,Y 492.138,Z 280.113,A -85,B 0,C 180,E1 -6407.082,E2 -6407.082} C_VEL
LIN {X 0,Y 492.063,Z 275.186,A -85,B 0,C 180,E1 -6407.256,E2 -6407.256} C_VEL
LIN {X 0,Y 489.076,Z 261.996,A -85,B 0,C 180,E1 -6407.713,E2 -6407.713} C_VEL
LIN {X 0,Y 488.127,Z 257.983,A -85,B 0,C 180,E1 -6407.822,E2 -6407.822} C_VEL
LIN {X 0,Y 488.178,Z 252.57,A -85,B 0,C 180,E1 -6411.095,E2 -6411.095} C_VEL
LIN {X 0,Y 488.255,Z 248.214,A -85,B 0,C 180,E1 -6413.768,E2 -6413.768} C_VEL
LIN {X 0,Y 488.326,Z 243.414,A -85,B 0,C 180,E1 -6416.835,E2 -6416.835} C_VEL
LIN {X 0,Y 488.436,Z 239.66,A -85,B 0,C 180,E1 -6419.289,E2 -6419.289} C_VEL
LIN {X 0,Y 488.557,Z 235.357,A -85,B 0,C 180,E1 -6422.158,E2 -6422.158} C_VEL
LIN {X 0,Y 488.719,Z 231.041,A -85,B 0,C 180,E1 -6425.115,E2 -6425.115} C_VEL
LIN {X 0,Y 488.718,Z 226.691,A -85,B 0,C 180,E1 -6428.197,E2 -6428.197} C_VEL
LIN {X 0,Y 488.637,Z 225.247,A -85,B 0,C 180,E1 -6429.261,E2 -6429.261} C_VEL
LIN {X 0,Y 488.7,Z 225.239,A -85,B 0,C 180,E1 -6431.598,E2 -6431.598} C_VEL
LIN {X 0,Y 488.715,Z 225.238,A -85,B 0,C 180,E1 -6434.801,E2 -6434.801} C_VEL
LIN {X 0,Y 488.673,Z 225.24,A -85,B 0,C 180,E1 -6437.472,E2 -6437.472} C_VEL
LIN {X 0,Y 488.696,Z 225.236,A -85,B 0,C 180,E1 -6440.745,E2 -6440.745} C_VEL
LIN {X 0,Y 488.68,Z 225.237,A -85,B 0,C 180,E1 -6443.868,E2 -6443.868} C_VEL
LIN {X 0,Y 488.738,Z 225.229,A -85,B 0,C 180,E1 -6446.877,E2 -6446.877} C_VEL
LIN {X 0,Y 488.722,Z 225.232,A -85,B 0,C 180,E1 -6449.78,E2 -6449.78} C_VEL
LIN {X 0,Y 488.794,Z 225.223,A -85,B 0,C 180,E1 -6453.057,E2 -6453.057} C_VEL
LIN {X 0,Y 488.683,Z 225.237,A -85,B 0,C 180,E1 -6456.254,E2 -6456.254} C_VEL
LIN {X 0,Y 488.75,Z 225.231,A -85,B 0,C 180,E1 -6459.176,E2 -6459.176} C_VEL
LIN {X 0,Y 488.751,Z 225.228,A -85,B 0,C 180,E1 -6461.632,E2 -6461.632} C_VEL
LIN {X 0,Y 488.764,Z 225.226,A -85,B 0,C 180,E1 -6465,E2 -6465} C_VEL
LIN {X 0,Y 488.809,Z 225.222,A -85,B 0,C 180,E1 -6468.388,E2 -6468.388} C_VEL
LIN {X 0,Y 488.788,Z 225.226,A -85,B 0,C 180,E1 -6471.733,E2 -6471.733} C_VEL
LIN {X 0,Y 488.851,Z 225.214,A -85,B 0,C 180,E1 -6474.224,E2 -6474.224} C_VEL
LIN {X 0,Y 488.953,Z 225.202,A -85,B 0,C 180,E1 -6477.529,E2 -6477.529} C_VEL
LIN {X 0,Y 488.937,Z 225.204,A -85,B 0,C 180,E1 -6480.824,E2 -6480.824} C_VEL
LIN {X 0,Y 488.964,Z 225.2,A -85,B 0,C 180,E1 -6482.471,E2 -6482.471} C_VEL
LIN {X 0,Y 488.832,Z 225.217,A -85,B 0,C 180,E1 -6485.776,E2 -6485.776} C_VEL
LIN {X 0,Y 488.765,Z 225.23,A -85,B 0,C 180,E1 -6488.267,E2 -6488.267} C_VEL
LIN {X 0,Y 488.809,Z 225.223,A -85,B 0,C 180,E1 -6491.612,E2 -6491.612} C_VEL
LIN {X 0,Y 488.768,Z 225.228,A -85,B 0,C 180,E1 -6495,E2 -6495} C_VEL
LIN {X 0,Y 488.747,Z 225.228,A -85,B 0,C 180,E1 -6498.442,E2 -6498.442} C_VEL
LIN {X 0,Y 488.71,Z 225.237,A -85,B 0,C 180,E1 -6501.071,E2 -6501.071} C_VEL
LIN {X 0,Y 488.678,Z 225.237,A -85,B 0,C 180,E1 -6503.746,E2 -6503.746} C_VEL
LIN {X 0,Y 488.703,Z 225.233,A -85,B 0,C 180,E1 -6506.922,E2 -6506.922} C_VEL
LIN {X 0,Y 488.721,Z 225.232,A -85,B 0,C 180,E1 -6510.219,E2 -6510.219} C_VEL
LIN {X 0,Y 488.737,Z 225.23,A -85,B 0,C 180,E1 -6513.484,E2 -6513.484} C_VEL
LIN {X 0,Y 488.675,Z 225.239,A -85,B 0,C 180,E1 -6516.353,E2 -6516.353} C_VEL
LIN {X 0,Y 488.702,Z 225.237,A -85,B 0,C 180,E1 -6519.254,E2 -6519.254} C_VEL
LIN {X 0,Y 488.71,Z 225.235,A -85,B 0,C 180,E1 -6521.6,E2 -6521.6} C_VEL
LIN {X 0,Y 488.703,Z 225.238,A -85,B 0,C 180,E1 -6524.803,E2 -6524.803} C_VEL
LIN {X 0,Y 488.67,Z 225.242,A -85,B 0,C 180,E1 -6527.472,E2 -6527.472} C_VEL
LIN {X 0,Y 488.759,Z 225.455,A -85,B 0,C 180,E1 -6528.725,E2 -6528.725} C_VEL
LIN {X 0,Y 489.285,Z 229.256,A -85,B 0,C 180,E1 -6530.864,E2 -6530.864} C_VEL
LIN {X 0,Y 489.32,Z 233.09,A -85,B 0,C 180,E1 -6532.898,E2 -6532.898} C_VEL
LIN {X 0,Y 489.133,Z 239.034,A -85,B 0,C 180,E1 -6535.919,E2 -6535.919} C_VEL
LIN {X 0,Y 488.978,Z 245.015,A -85,B 0,C 180,E1 -6538.84,E2 -6538.84} C_VEL
LIN {X 0,Y 488.753,Z 252.022,A -85,B 0,C 180,E1 -6542.139,E2 -6542.139} C_VEL
LIN {X 0,Y 488.514,Z 259.05,A -85,B 0,C 180,E1 -6545.341,E2 -6545.341} C_VEL
LIN {X 0,Y 488.354,Z 265.007,A -85,B 0,C 180,E1 -6548.027,E2 -6548.027} C_VEL
LIN {X 0,Y 488.235,Z 270.956,A -85,B 0,C 180,E1 -6550.666,E2 -6550.666} C_VEL
LIN {X 0,Y 488.133,Z 274.467,A -85,B 0,C 180,E1 -6552.2,E2 -6552.2} C_VEL
LIN {X 0,Y 491.259,Z 289.628,A -85,B 0,C 180,E1 -6552.661,E2 -6552.661} C_VEL
LIN {X 0,Y 492.144,Z 295.393,A -85,B 0,C 180,E1 -6552.873,E2 -6552.873} C_VEL
LIN {X 0,Y 491.739,Z 308.659,A -85,B 0,C 180,E1 -6553.391,E2 -6553.391} C_VEL
LIN {X 0,Y 491.141,Z 322.614,A -85,B 0,C 180,E1 -6554.117,E2 -6554.117} C_VEL
LIN {X 0,Y 490.578,Z 335.101,A -85,B 0,C 180,E1 -6554.95,E2 -6554.95} C_VEL
LIN {X 0,Y 490.006,Z 347.687,A -85,B 0,C 180,E1 -6555.993,E2 -6555.993} C_VEL
LIN {X 0,Y 489.445,Z 358.9,A -85,B 0,C 180,E1 -6557.14,E2 -6557.14} C_VEL
LIN {X 0,Y 489.041,Z 368.959,A -85,B 0,C 180,E1 -6558.393,E2 -6558.393} C_VEL
LIN {X 0,Y 488.622,Z 377.311,A -85,B 0,C 180,E1 -6559.642,E2 -6559.642} C_VEL
LIN {X 0,Y 488.332,Z 385.298,A -85,B 0,C 180,E1 -6561.1,E2 -6561.1} C_VEL
LIN {X 0,Y 488.107,Z 391.73,A -85,B 0,C 180,E1 -6562.554,E2 -6562.554} C_VEL
LIN {X 0,Y 488.021,Z 396.167,A -85,B 0,C 180,E1 -6563.793,E2 -6563.793} C_VEL
LIN {X 0,Y 487.96,Z 399.686,A -85,B 0,C 180,E1 -6565.042,E2 -6565.042} C_VEL
LIN {X 0,Y 487.955,Z 403.094,A -85,B 0,C 180,E1 -6566.697,E2 -6566.697} C_VEL
LIN {X 0,Y 487.886,Z 405.108,A -85,B 0,C 180,E1 -6568.349,E2 -6568.349} C_VEL
LIN {X 0,Y 487.817,Z 405.776,A -85,B 0,C 180,E1 -6570,E2 -6570} C_VEL
LIN {X 0,Y 487.886,Z 405.11,A -85,B 0,C 180,E1 -6571.651,E2 -6571.651} C_VEL
LIN {X 0,Y 487.955,Z 403.098,A -85,B 0,C 180,E1 -6573.303,E2 -6573.303} C_VEL
LIN {X 0,Y 487.96,Z 399.69,A -85,B 0,C 180,E1 -6574.957,E2 -6574.957} C_VEL
LIN {X 0,Y 488.042,Z 394.785,A -85,B 0,C 180,E1 -6576.615,E2 -6576.615} C_VEL
LIN {X 0,Y 488.238,Z 388.24,A -85,B 0,C 180,E1 -6578.276,E2 -6578.276} C_VEL
LIN {X 0,Y 488.503,Z 380.958,A -85,B 0,C 180,E1 -6579.732,E2 -6579.732} C_VEL
LIN {X 0,Y 488.909,Z 371.94,A -85,B 0,C 180,E1 -6581.19,E2 -6581.19} C_VEL
LIN {X 0,Y 489.346,Z 362.477,A -85,B 0,C 180,E1 -6582.441,E2 -6582.441} C_VEL
LIN {X 0,Y 489.787,Z 352.002,A -85,B 0,C 180,E1 -6583.59,E2 -6583.59} C_VEL
LIN {X 0,Y 490.329,Z 340.445,A -85,B 0,C 180,E1 -6584.633,E2 -6584.633} C_VEL
LIN {X 0,Y 490.863,Z 329.212,A -85,B 0,C 180,E1 -6585.466,E2 -6585.466} C_VEL
LIN {X 0,Y 491.409,Z 317.102,A -85,B 0,C 180,E1 -6586.194,E2 -6586.194} C_VEL
LIN {X 0,Y 491.846,Z 303.798,A -85,B 0,C 180,E1 -6586.819,E2 -6586.819} C_VEL
LIN {X 0,Y 492.004,Z 293.487,A -85,B 0,C 180,E1 -6587.198,E2 -6587.198} C_VEL
LIN {X 0,Y 489.128,Z 279.14,A -85,B 0,C 180,E1 -6587.676,E2 -6587.676} C_VEL
LIN {X 0,Y 488.132,Z 274.467,A -85,B 0,C 180,E1 -6587.799,E2 -6587.799} C_VEL
LIN {X 0,Y 488.328,Z 267.873,A -85,B 0,C 180,E1 -6590.695,E2 -6590.695} C_VEL
LIN {X 0,Y 488.445,Z 261.04,A -85,B 0,C 180,E1 -6593.758,E2 -6593.758} C_VEL
LIN {X 0,Y 488.694,Z 254.052,A -85,B 0,C 180,E1 -6596.921,E2 -6596.921} C_VEL
LIN {X 0,Y 488.891,Z 247,A -85,B 0,C 180,E1 -6600.208,E2 -6600.208} C_VEL
LIN {X 0,Y 489.081,Z 241.015,A -85,B 0,C 180,E1 -6603.097,E2 -6603.097} C_VEL
LIN {X 0,Y 489.258,Z 235.05,A -85,B 0,C 180,E1 -6606.082,E2 -6606.082} C_VEL
LIN {X 0,Y 489.361,Z 231.089,A -85,B 0,C 180,E1 -6608.137,E2 -6608.137} C_VEL
LIN {X 0,Y 489.025,Z 226.988,A -85,B 0,C 180,E1 -6610.387,E2 -6610.387} C_VEL
LIN {X 0,Y 488.715,Z 225.235,A -85,B 0,C 180,E1 -6611.415,E2 -6611.415} C_VEL
LIN {X 0,Y 488.702,Z 225.24,A -85,B 0,C 180,E1 -6614.803,E2 -6614.803} C_VEL
LIN {X 0,Y 488.693,Z 225.239,A -85,B 0,C 180,E1 -6617.475,E2 -6617.475} C_VEL
LIN {X 0,Y 488.734,Z 225.234,A -85,B 0,C 180,E1 -6619.677,E2 -6619.677} C_VEL
LIN {X 0,Y 488.671,Z 225.243,A -85,B 0,C 180,E1 -6622.84,E2 -6622.84} C_VEL
LIN {X 0,Y 488.731,Z 225.236,A -85,B 0,C 180,E1 -6625.887,E2 -6625.887} C_VEL
LIN {X 0,Y 488.693,Z 225.237,A -85,B 0,C 180,E1 -6628.82,E2 -6628.82} C_VEL
LIN {X 0,Y 488.699,Z 225.234,A -85,B 0,C 180,E1 -6631.668,E2 -6631.668} C_VEL
LIN {X 0,Y 488.702,Z 225.235,A -85,B 0,C 180,E1 -6634.442,E2 -6634.442} C_VEL
LIN {X 0,Y 488.724,Z 225.235,A -85,B 0,C 180,E1 -6637.153,E2 -6637.153} C_VEL
LIN {X 0,Y 488.725,Z 225.231,A -85,B 0,C 180,E1 -6639.81,E2 -6639.81} C_VEL
LIN {X 0,Y 488.701,Z 225.236,A -85,B 0,C 180,E1 -6642.422,E2 -6642.422} C_VEL
LIN {X 0,Y 488.767,Z 225.227,A -85,B 0,C 180,E1 -6645,E2 -6645} C_VEL
LIN {X 0,Y 488.808,Z 225.223,A -85,B 0,C 180,E1 -6648.388,E2 -6648.388} C_VEL
LIN {X 0,Y 488.763,Z 225.23,A -85,B 0,C 180,E1 -6651.733,E2 -6651.733} C_VEL
LIN {X 0,Y 488.83,Z 225.217,A -85,B 0,C 180,E1 -6654.224,E2 -6654.224} C_VEL
LIN {X 0,Y 488.963,Z 225.201,A -85,B 0,C 180,E1 -6657.529,E2 -6657.529} C_VEL
LIN {X 0,Y 488.97,Z 225.205,A -85,B 0,C 180,E1 -6660,E2 -6660} C_VEL
LIN {X 0,Y 488.951,Z 225.202,A -85,B 0,C 180,E1 -6662.471,E2 -6662.471} C_VEL
LIN {X 0,Y 488.849,Z 225.215,A -85,B 0,C 180,E1 -6665.776,E2 -6665.776} C_VEL
LIN {X 0,Y 488.819,Z 225.222,A -85,B 0,C 180,E1 -6668.266,E2 -6668.266} C_VEL
LIN {X 0,Y 488.808,Z 225.223,A -85,B 0,C 180,E1 -6671.612,E2 -6671.612} C_VEL
LIN {X 0,Y 488.762,Z 225.227,A -85,B 0,C 180,E1 -6675,E2 -6675} C_VEL
LIN {X 0,Y 488.758,Z 225.227,A -85,B 0,C 180,E1 -6678.442,E2 -6678.442} C_VEL
LIN {X 0,Y 488.708,Z 225.238,A -85,B 0,C 180,E1 -6681.071,E2 -6681.071} C_VEL
LIN {X 0,Y 488.681,Z 225.236,A -85,B 0,C 180,E1 -6683.746,E2 -6683.746} C_VEL
LIN {X 0,Y 488.793,Z 225.222,A -85,B 0,C 180,E1 -6686.943,E2 -6686.943} C_VEL
LIN {X 0,Y 488.71,Z 225.234,A -85,B 0,C 180,E1 -6690.363,E2 -6690.363} C_VEL
LIN {X 0,Y 488.731,Z 225.231,A -85,B 0,C 180,E1 -6693.483,E2 -6693.483} C_VEL
LIN {X 0,Y 488.684,Z 225.236,A -85,B 0,C 180,E1 -6696.355,E2 -6696.355} C_VEL
LIN {X 0,Y 488.695,Z 225.236,A -85,B 0,C 180,E1 -6699.255,E2 -6699.255} C_VEL
LIN {X 0,Y 488.672,Z 225.24,A -85,B 0,C 180,E1 -6702.528,E2 -6702.528} C_VEL
LIN {X 0,Y 488.703,Z 225.238,A -85,B 0,C 180,E1 -6705.197,E2 -6705.197} C_VEL
LIN {X 0,Y 488.699,Z 225.239,A -85,B 0,C 180,E1 -6708.402,E2 -6708.402} C_VEL
LIN {X 0,Y 488.689,Z 225.39,A -85,B 0,C 180,E1 -6710.95,E2 -6710.95} C_VEL
LIN {X 0,Y 488.72,Z 229.456,A -85,B 0,C 180,E1 -6713.872,E2 -6713.872} C_VEL
LIN {X 0,Y 488.625,Z 233.294,A -85,B 0,C 180,E1 -6716.536,E2 -6716.536} C_VEL
LIN {X 0,Y 488.472,Z 238.082,A -85,B 0,C 180,E1 -6719.763,E2 -6719.763} C_VEL
LIN {X 0,Y 488.338,Z 242.361,A -85,B 0,C 180,E1 -6722.578,E2 -6722.578} C_VEL
LIN {X 0,Y 488.284,Z 244.704,A -85,B 0,C 180,E1 -6724.093,E2 -6724.093} C_VEL
LIN {X 0,Y 487.603,Z 245.825,A -85,B 0,C 180,E1 -6724.769,E2 -6724.769} C_VEL
LIN {X 0,Y 484.71,Z 247.833,A -85,B 0,C 180,E1 -6725.86,E2 -6725.86} C_VEL
LIN {X 0,Y 482.265,Z 249.468,A -85,B 0,C 180,E1 -6726.739,E2 -6726.739} C_VEL
LIN {X 0,Y 481.213,Z 250.657,A -85,B 0,C 180,E1 -6727.42,E2 -6727.42} C_VEL
LIN {X 0,Y 481.126,Z 251.036,A -85,B 0,C 180,E1 -6727.652,E2 -6727.652} C_VEL
LIN {X 0,Y 481.059,Z 255.435,A -85,B 0,C 180,E1 -6730.366,E2 -6730.366} C_VEL
LIN {X 0,Y 481.05,Z 258.102,A -85,B 0,C 180,E1 -6731.993,E2 -6731.993} C_VEL
LIN {X 0,Y 484.66,Z 273.117,A -85,B 0,C 180,E1 -6732.497,E2 -6732.497} C_VEL
LIN {X 0,Y 485.454,Z 277.711,A -85,B 0,C 180,E1 -6732.677,E2 -6732.677} C_VEL
LIN {X 0,Y 485.058,Z 291.084,A -85,B 0,C 180,E1 -6733.209,E2 -6733.209} C_VEL
LIN {X 0,Y 484.564,Z 304.081,A -85,B 0,C 180,E1 -6733.896,E2 -6733.896} C_VEL
LIN {X 0,Y 483.949,Z 316.66,A -85,B 0,C 180,E1 -6734.739,E2 -6734.739} C_VEL
LIN {X 0,Y 483.361,Z 328.115,A -85,B 0,C 180,E1 -6735.689,E2 -6735.689} C_VEL
LIN {X 0,Y 482.809,Z 338.625,A -85,B 0,C 180,E1 -6736.746,E2 -6736.746} C_VEL
LIN {X 0,Y 482.338,Z 348.14,A -85,B 0,C 180,E1 -6737.896,E2 -6737.896} C_VEL
LIN {X 0,Y 481.826,Z 357.657,A -85,B 0,C 180,E1 -6739.282,E2 -6739.282} C_VEL
LIN {X 0,Y 481.458,Z 365.902,A -85,B 0,C 180,E1 -6740.76,E2 -6740.76} C_VEL
LIN {X 0,Y 481.206,Z 371.645,A -85,B 0,C 180,E1 -6742.025,E2 -6742.025} C_VEL
LIN {X 0,Y 481.045,Z 376.915,A -85,B 0,C 180,E1 -6743.451,E2 -6743.451} C_VEL
LIN {X 0,Y 480.902,Z 381.261,A -85,B 0,C 180,E1 -6744.97,E2 -6744.97} C_VEL
LIN {X 0,Y 480.888,Z 384.666,A -85,B 0,C 180,E1 -6746.649,E2 -6746.649} C_VEL
LIN {X 0,Y 480.791,Z 386.693,A -85,B 0,C 180,E1 -6748.325,E2 -6748.325} C_VEL
LIN {X 0,Y 480.741,Z 387.393,A -85,B 0,C 180,E1 -6750,E2 -6750} C_VEL
LIN {X 0,Y 480.789,Z 386.772,A -85,B 0,C 180,E1 -6751.675,E2 -6751.675} C_VEL
LIN {X 0,Y 480.887,Z 384.817,A -85,B 0,C 180,E1 -6753.351,E2 -6753.351} C_VEL
LIN {X 0,Y 480.9,Z 381.484,A -85,B 0,C 180,E1 -6755.031,E2 -6755.031} C_VEL
LIN {X 0,Y 481.075,Z 377.112,A -85,B 0,C 180,E1 -6756.58,E2 -6756.58} C_VEL
LIN {X 0,Y 481.198,Z 372.029,A -85,B 0,C 180,E1 -6757.976,E2 -6757.976} C_VEL
LIN {X 0,Y 481.483,Z 365.273,A -85,B 0,C 180,E1 -6759.452,E2 -6759.452} C_VEL
LIN {X 0,Y 481.87,Z 356.879,A -85,B 0,C 180,E1 -6760.93,E2 -6760.93} C_VEL
LIN {X 0,Y 482.314,Z 348.861,A -85,B 0,C 180,E1 -6762.1,E2 -6762.1} C_VEL
LIN {X 0,Y 482.744,Z 339.443,A -85,B 0,C 180,E1 -6763.256,E2 -6763.256} C_VEL
LIN {X 0,Y 483.393,Z 327.927,A -85,B 0,C 180,E1 -6764.417,E2 -6764.417} C_VEL
LIN {X 0,Y 483.98,Z 316.424,A -85,B 0,C 180,E1 -6765.368,E2 -6765.368} C_VEL
LIN {X 0,Y 484.551,Z 303.791,A -85,B 0,C 180,E1 -6766.213,E2 -6766.213} C_VEL
LIN {X 0,Y 485.063,Z 290.721,A -85,B 0,C 180,E1 -6766.899,E2 -6766.899} C_VEL
LIN {X 0,Y 485.314,Z 276.59,A -85,B 0,C 180,E1 -6767.46,E2 -6767.46} C_VEL
LIN {X 0,Y 482.243,Z 262.943,A -85,B 0,C 180,E1 -6767.955,E2 -6767.955} C_VEL
LIN {X 0,Y 481.056,Z 258.074,A -85,B 0,C 180,E1 -6768.115,E2 -6768.115} C_VEL
LIN {X 0,Y 481.095,Z 252.678,A -85,B 0,C 180,E1 -6771.421,E2 -6771.421} C_VEL
LIN {X 0,Y 481.208,Z 248.319,A -85,B 0,C 180,E1 -6774.138,E2 -6774.138} C_VEL
LIN {X 0,Y 481.264,Z 243.865,A -85,B 0,C 180,E1 -6777.026,E2 -6777.026} C_VEL
LIN {X 0,Y 481.403,Z 239.751,A -85,B 0,C 180,E1 -6779.76,E2 -6779.76} C_VEL
LIN {X 0,Y 481.517,Z 235.438,A -85,B 0,C 180,E1 -6782.686,E2 -6782.686} C_VEL
LIN {X 0,Y 481.67,Z 231.818,A -85,B 0,C 180,E1 -6785.205,E2 -6785.205} C_VEL
LIN {X 0,Y 481.693,Z 227.896,A -85,B 0,C 180,E1 -6788.013,E2 -6788.013} C_VEL
LIN {X 0,Y 481.606,Z 226.124,A -85,B 0,C 180,E1 -6789.338,E2 -6789.338} C_VEL
LIN {X 0,Y 481.647,Z 226.114,A -85,B 0,C 180,E1 -6792.161,E2 -6792.161} C_VEL
LIN {X 0,Y 481.662,Z 226.112,A -85,B 0,C 180,E1 -6795.543,E2 -6795.543} C_VEL
LIN {X 0,Y 481.634,Z 226.116,A -85,B 0,C 180,E1 -6798.956,E2 -6798.956} C_VEL
LIN {X 0,Y 481.655,Z 226.111,A -85,B 0,C 180,E1 -6801.993,E2 -6801.993} C_VEL
LIN {X 0,Y 481.688,Z 226.108,A -85,B 0,C 180,E1 -6805.318,E2 -6805.318} C_VEL
LIN {X 0,Y 481.646,Z 226.113,A -85,B 0,C 180,E1 -6808.311,E2 -6808.311} C_VEL
LIN {X 0,Y 481.7,Z 226.108,A -85,B 0,C 180,E1 -6811.218,E2 -6811.218} C_VEL
LIN {X 0,Y 481.693,Z 226.112,A -85,B 0,C 180,E1 -6814.042,E2 -6814.042} C_VEL
LIN {X 0,Y 481.677,Z 226.109,A -85,B 0,C 180,E1 -6816.812,E2 -6816.812} C_VEL
LIN {X 0,Y 481.698,Z 226.106,A -85,B 0,C 180,E1 -6819.503,E2 -6819.503} C_VEL
LIN {X 0,Y 481.692,Z 226.111,A -85,B 0,C 180,E1 -6822.158,E2 -6822.158} C_VEL
LIN {X 0,Y 481.746,Z 226.1,A -85,B 0,C 180,E1 -6824.776,E2 -6824.776} C_VEL
LIN {X 0,Y 481.754,Z 226.1,A -85,B 0,C 180,E1 -6828.215,E2 -6828.215} C_VEL
LIN {X 0,Y 481.743,Z 226.102,A -85,B 0,C 180,E1 -6831.611,E2 -6831.611} C_VEL
LIN {X 0,Y 481.811,Z 226.092,A -85,B 0,C 180,E1 -6834.139,E2 -6834.139} C_VEL
LIN {X 0,Y 481.919,Z 226.078,A -85,B 0,C 180,E1 -6837.492,E2 -6837.492} C_VEL
LIN {X 0,Y 481.889,Z 226.082,A -85,B 0,C 180,E1 -6840.836,E2 -6840.836} C_VEL
LIN {X 0,Y 481.931,Z 226.076,A -85,B 0,C 180,E1 -6842.507,E2 -6842.507} C_VEL
LIN {X 0,Y 481.791,Z 226.094,A -85,B 0,C 180,E1 -6845.861,E2 -6845.861} C_VEL
LIN {X 0,Y 481.724,Z 226.106,A -85,B 0,C 180,E1 -6848.389,E2 -6848.389} C_VEL
LIN {X 0,Y 481.754,Z 226.1,A -85,B 0,C 180,E1 -6851.785,E2 -6851.785} C_VEL
LIN {X 0,Y 481.747,Z 226.101,A -85,B 0,C 180,E1 -6855.224,E2 -6855.224} C_VEL
LIN {X 0,Y 481.709,Z 226.105,A -85,B 0,C 180,E1 -6858.722,E2 -6858.722} C_VEL
LIN {X 0,Y 481.649,Z 226.115,A -85,B 0,C 180,E1 -6861.395,E2 -6861.395} C_VEL
LIN {X 0,Y 481.656,Z 226.114,A -85,B 0,C 180,E1 -6864.114,E2 -6864.114} C_VEL
LIN {X 0,Y 481.657,Z 226.112,A -85,B 0,C 180,E1 -6867.117,E2 -6867.117} C_VEL
LIN {X 0,Y 481.669,Z 226.111,A -85,B 0,C 180,E1 -6869.742,E2 -6869.742} C_VEL
LIN {X 0,Y 481.675,Z 226.112,A -85,B 0,C 180,E1 -6872.674,E2 -6872.674} C_VEL
LIN {X 0,Y 481.662,Z 226.113,A -85,B 0,C 180,E1 -6875.204,E2 -6875.204} C_VEL
LIN {X 0,Y 481.672,Z 226.115,A -85,B 0,C 180,E1 -6878.859,E2 -6878.859} C_VEL
LIN {X 0,Y 481.655,Z 226.116,A -85,B 0,C 180,E1 -6881.913,E2 -6881.913} C_VEL
LIN {X 0,Y 481.656,Z 226.116,A -85,B 0,C 180,E1 -6884.458,E2 -6884.458} C_VEL
LIN {X 0,Y 481.639,Z 226.117,A -85,B 0,C 180,E1 -6887.838,E2 -6887.838} C_VEL
LIN {X 0,Y 481.673,Z 226.14,A -85,B 0,C 180,E1 -6888.403,E2 -6888.403} C_VEL
LIN {X 0,Y 482.225,Z 229.93,A -85,B 0,C 180,E1 -6890.572,E2 -6890.572} C_VEL
LIN {X 0,Y 482.354,Z 233.034,A -85,B 0,C 180,E1 -6892.269,E2 -6892.269} C_VEL
LIN {X 0,Y 482.13,Z 238.966,A -85,B 0,C 180,E1 -6895.354,E2 -6895.354} C_VEL
LIN {X 0,Y 481.968,Z 244.937,A -85,B 0,C 180,E1 -6898.335,E2 -6898.335} C_VEL
LIN {X 0,Y 481.762,Z 250.935,A -85,B 0,C 180,E1 -6901.222,E2 -6901.222} C_VEL
LIN {X 0,Y 481.529,Z 256.941,A -85,B 0,C 180,E1 -6904.033,E2 -6904.033} C_VEL
LIN {X 0,Y 481.365,Z 263.167,A -85,B 0,C 180,E1 -6906.898,E2 -6906.898} C_VEL
LIN {X 0,Y 481.226,Z 268.852,A -85,B 0,C 180,E1 -6909.482,E2 -6909.482} C_VEL
LIN {X 0,Y 481.092,Z 274.471,A -85,B 0,C 180,E1 -6911.936,E2 -6911.936} C_VEL
LIN {X 0,Y 484.129,Z 289.097,A -85,B 0,C 180,E1 -6912.386,E2 -6912.386} C_VEL
LIN {X 0,Y 485.314,Z 296.101,A -85,B 0,C 180,E1 -6912.654,E2 -6912.654} C_VEL
LIN {X 0,Y 484.866,Z 309.929,A -85,B 0,C 180,E1 -6913.215,E2 -6913.215} C_VEL
LIN {X 0,Y 484.284,Z 322.519,A -85,B 0,C 180,E1 -6913.888,E2 -6913.888} C_VEL
LIN {X 0,Y 483.668,Z 334.966,A -85,B 0,C 180,E1 -6914.73,E2 -6914.73} C_VEL
LIN {X 0,Y 483.088,Z 347.553,A -85,B 0,C 180,E1 -6915.789,E2 -6915.789} C_VEL
LIN {X 0,Y 482.478,Z 358.765,A -85,B 0,C 180,E1 -6916.951,E2 -6916.951} C_VEL
LIN {X 0,Y 482.036,Z 368.823,A -85,B 0,C 180,E1 -6918.222,E2 -6918.222} C_VEL
LIN {X 0,Y 481.599,Z 377.176,A -85,B 0,C 180,E1 -6919.49,E2 -6919.49} C_VEL
LIN {X 0,Y 481.283,Z 385.163,A -85,B 0,C 180,E1 -6920.968,E2 -6920.968} C_VEL
LIN {X 0,Y 481.026,Z 391.594,A -85,B 0,C 180,E1 -6922.444,E2 -6922.444} C_VEL
LIN {X 0,Y 480.965,Z 395.486,A -85,B 0,C 180,E1 -6923.533,E2 -6923.533} C_VEL
LIN {X 0,Y 480.891,Z 399.552,A -85,B 0,C 180,E1 -6924.969,E2 -6924.969} C_VEL
LIN {X 0,Y 480.861,Z 402.959,A -85,B 0,C 180,E1 -6926.648,E2 -6926.648} C_VEL
LIN {X 0,Y 480.787,Z 404.974,A -85,B 0,C 180,E1 -6928.325,E2 -6928.325} C_VEL
LIN {X 0,Y 480.741,Z 405.641,A -85,B 0,C 180,E1 -6930,E2 -6930} C_VEL
LIN {X 0,Y 480.787,Z 404.975,A -85,B 0,C 180,E1 -6931.675,E2 -6931.675} C_VEL
LIN {X 0,Y 480.861,Z 402.963,A -85,B 0,C 180,E1 -6933.351,E2 -6933.351} C_VEL
LIN {X 0,Y 480.891,Z 399.555,A -85,B 0,C 180,E1 -6935.031,E2 -6935.031} C_VEL
LIN {X 0,Y 480.962,Z 394.65,A -85,B 0,C 180,E1 -6936.713,E2 -6936.713} C_VEL
LIN {X 0,Y 481.159,Z 388.104,A -85,B 0,C 180,E1 -6938.399,E2 -6938.399} C_VEL
LIN {X 0,Y 481.454,Z 380.822,A -85,B 0,C 180,E1 -6939.876,E2 -6939.876} C_VEL
LIN {X 0,Y 481.906,Z 371.805,A -85,B 0,C 180,E1 -6941.355,E2 -6941.355} C_VEL
LIN {X 0,Y 482.359,Z 362.341,A -85,B 0,C 180,E1 -6942.624,E2 -6942.624} C_VEL
LIN {X 0,Y 482.839,Z 351.865,A -85,B 0,C 180,E1 -6943.789,E2 -6943.789} C_VEL
LIN {X 0,Y 483.406,Z 340.308,A -85,B 0,C 180,E1 -6944.847,E2 -6944.847} C_VEL
LIN {X 0,Y 484.06,Z 327.49,A -85,B 0,C 180,E1 -6945.797,E2 -6945.797} C_VEL
LIN {X 0,Y 484.644,Z 315.452,A -85,B 0,C 180,E1 -6946.508,E2 -6946.508} C_VEL
LIN {X 0,Y 485.068,Z 302.357,A -85,B 0,C 180,E1 -6947.115,E2 -6947.115} C_VEL
LIN {X 0,Y 485.137,Z 294.384,A -85,B 0,C 180,E1 -6947.412,E2 -6947.412} C_VEL
LIN {X 0,Y 482.31,Z 280.226,A -85,B 0,C 180,E1 -6947.909,E2 -6947.909} C_VEL
LIN {X 0,Y 481.065,Z 274.342,A -85,B 0,C 180,E1 -6948.068,E2 -6948.068} C_VEL
LIN {X 0,Y 481.257,Z 268.146,A -85,B 0,C 180,E1 -6950.833,E2 -6950.833} C_VEL
LIN {X 0,Y 481.409,Z 260.937,A -85,B 0,C 180,E1 -6954.127,E2 -6954.127} C_VEL
LIN {X 0,Y 481.662,Z 254.441,A -85,B 0,C 180,E1 -6957.119,E2 -6957.119} C_VEL
LIN {X 0,Y 481.84,Z 248.918,A -85,B 0,C 180,E1 -6959.73,E2 -6959.73} C_VEL
LIN {X 0,Y 482.007,Z 242.932,A -85,B 0,C 180,E1 -6962.649,E2 -6962.649} C_VEL
LIN {X 0,Y 482.213,Z 236.966,A -85,B 0,C 180,E1 -6965.66,E2 -6965.66} C_VEL
LIN {X 0,Y 482.372,Z 232.292,A -85,B 0,C 180,E1 -6968.116,E2 -6968.116} C_VEL
LIN {X 0,Y 481.977,Z 227.664,A -85,B 0,C 180,E1 -6970.69,E2 -6970.69} C_VEL
LIN {X 0,Y 481.66,Z 226.114,A -85,B 0,C 180,E1 -6971.676,E2 -6971.676} C_VEL
LIN {X 0,Y 481.654,Z 226.115,A -85,B 0,C 180,E1 -6974.458,E2 -6974.458} C_VEL
LIN {X 0,Y 481.649,Z 226.117,A -85,B 0,C 180,E1 -6977.839,E2 -6977.839} C_VEL
LIN {X 0,Y 481.662,Z 226.113,A -85,B 0,C 180,E1 -6980.654,E2 -6980.654} C_VEL
LIN {X 0,Y 481.622,Z 226.117,A -85,B 0,C 180,E1 -6983.377,E2 -6983.377} C_VEL
LIN {X 0,Y 481.711,Z 226.107,A -85,B 0,C 180,E1 -6986.33,E2 -6986.33} C_VEL
LIN {X 0,Y 481.651,Z 226.115,A -85,B 0,C 180,E1 -6989.418,E2 -6989.418} C_VEL
LIN {X 0,Y 481.657,Z 226.114,A -85,B 0,C 180,E1 -6992.165,E2 -6992.165} C_VEL
LIN {X 0,Y 481.679,Z 226.109,A -85,B 0,C 180,E1 -6994.968,E2 -6994.968} C_VEL
LIN {X 0,Y 481.651,Z 226.114,A -85,B 0,C 180,E1 -6997.705,E2 -6997.705} C_VEL
LIN {X 0,Y 481.702,Z 226.11,A -85,B 0,C 180,E1 -7000.393,E2 -7000.393} C_VEL
LIN {X 0,Y 481.667,Z 226.109,A -85,B 0,C 180,E1 -7003.033,E2 -7003.033} C_VEL
LIN {X 0,Y 481.696,Z 226.108,A -85,B 0,C 180,E1 -7005.639,E2 -7005.639} C_VEL
LIN {X 0,Y 481.753,Z 226.1,A -85,B 0,C 180,E1 -7008.215,E2 -7008.215} C_VEL
LIN {X 0,Y 481.722,Z 226.106,A -85,B 0,C 180,E1 -7011.611,E2 -7011.611} C_VEL
LIN {X 0,Y 481.789,Z 226.095,A -85,B 0,C 180,E1 -7014.139,E2 -7014.139} C_VEL
LIN {X 0,Y 481.93,Z 226.077,A -85,B 0,C 180,E1 -7017.493,E2 -7017.493} C_VEL
LIN {X 0,Y 481.94,Z 226.081,A -85,B 0,C 180,E1 -7020,E2 -7020} C_VEL
LIN {X 0,Y 481.918,Z 226.078,A -85,B 0,C 180,E1 -7022.508,E2 -7022.508} C_VEL
LIN {X 0,Y 481.81,Z 226.092,A -85,B 0,C 180,E1 -7025.861,E2 -7025.861} C_VEL
LIN {X 0,Y 481.764,Z 226.1,A -85,B 0,C 180,E1 -7028.388,E2 -7028.388} C_VEL
LIN {X 0,Y 481.753,Z 226.1,A -85,B 0,C 180,E1 -7031.785,E2 -7031.785} C_VEL
LIN {X 0,Y 481.744,Z 226.1,A -85,B 0,C 180,E1 -7035.224,E2 -7035.224} C_VEL
LIN {X 0,Y 481.714,Z 226.104,A -85,B 0,C 180,E1 -7038.722,E2 -7038.722} C_VEL
LIN {X 0,Y 481.647,Z 226.114,A -85,B 0,C 180,E1 -7041.395,E2 -7041.395} C_VEL
LIN {X 0,Y 481.662,Z 226.114,A -85,B 0,C 180,E1 -7044.114,E2 -7044.114} C_VEL
LIN {X 0,Y 481.748,Z 226.101,A -85,B 0,C 180,E1 -7047.139,E2 -7047.139} C_VEL
LIN {X 0,Y 481.679,Z 226.109,A -85,B 0,C 180,E1 -7049.741,E2 -7049.741} C_VEL
LIN {X 0,Y 481.672,Z 226.112,A -85,B 0,C 180,E1 -7052.674,E2 -7052.674} C_VEL
LIN {X 0,Y 481.638,Z 226.119,A -85,B 0,C 180,E1 -7055.71,E2 -7055.71} C_VEL
LIN {X 0,Y 481.668,Z 226.115,A -85,B 0,C 180,E1 -7058.86,E2 -7058.86} C_VEL
LIN {X 0,Y 481.632,Z 226.12,A -85,B 0,C 180,E1 -7062.163,E2 -7062.163} C_VEL
LIN {X 0,Y 481.656,Z 226.116,A -85,B 0,C 180,E1 -7065.542,E2 -7065.542} C_VEL
LIN {X 0,Y 481.643,Z 226.117,A -85,B 0,C 180,E1 -7068.957,E2 -7068.957} C_VEL
LIN {X 0,Y 481.648,Z 226.117,A -85,B 0,C 180,E1 -7070.656,E2 -7070.656} C_VEL
LIN {X 0,Y 481.697,Z 229.68,A -85,B 0,C 180,E1 -7073.365,E2 -7073.365} C_VEL
LIN {X 0,Y 481.605,Z 233.854,A -85,B 0,C 180,E1 -7076.322,E2 -7076.322} C_VEL
LIN {X 0,Y 481.446,Z 238.439,A -85,B 0,C 180,E1 -7079.459,E2 -7079.459} C_VEL
LIN {X 0,Y 481.306,Z 242.453,A -85,B 0,C 180,E1 -7082.143,E2 -7082.143} C_VEL
LIN {X 0,Y 481.235,Z 246.735,A -85,B 0,C 180,E1 -7084.943,E2 -7084.943} C_VEL
LIN {X 0,Y 481.126,Z 251.036,A -85,B 0,C 180,E1 -7087.652,E2 -7087.652} C_VEL
LIN {X 0,Y 480.446,Z 252.203,A -85,B 0,C 180,E1 -7088.336,E2 -7088.336} C_VEL
LIN {X 0,Y 477.554,Z 254.252,A -85,B 0,C 180,E1 -7089.444,E2 -7089.444} C_VEL
LIN {X 0,Y 475.108,Z 255.906,A -85,B 0,C 180,E1 -7090.336,E2 -7090.336} C_VEL
LIN {X 0,Y 474.055,Z 257.112,A -85,B 0,C 180,E1 -7091.028,E2 -7091.028} C_VEL
LIN {X 0,Y 473.968,Z 257.499,A -85,B 0,C 180,E1 -7091.262,E2 -7091.262} C_VEL
LIN {X 0,Y 473.975,Z 258.217,A -85,B 0,C 180,E1 -7091.705,E2 -7091.705} C_VEL
LIN {X 0,Y 477.861,Z 274.282,A -85,B 0,C 180,E1 -7092.271,E2 -7092.271} C_VEL
LIN {X 0,Y 478.658,Z 278.764,A -85,B 0,C 180,E1 -7092.455,E2 -7092.455} C_VEL
LIN {X 0,Y 478.228,Z 292.357,A -85,B 0,C 180,E1 -7093.017,E2 -7093.017} C_VEL
LIN {X 0,Y 477.615,Z 305.988,A -85,B 0,C 180,E1 -7093.765,E2 -7093.765} C_VEL
LIN {X 0,Y 477.015,Z 318.224,A -85,B 0,C 180,E1 -7094.621,E2 -7094.621} C_VEL
LIN {X 0,Y 476.359,Z 330.558,A -85,B 0,C 180,E1 -7095.693,E2 -7095.693} C_VEL
LIN {X 0,Y 475.738,Z 340.688,A -85,B 0,C 180,E1 -7096.763,E2 -7096.763} C_VEL
LIN {X 0,Y 475.257,Z 350.737,A -85,B 0,C 180,E1 -7098.052,E2 -7098.052} C_VEL
LIN {X 0,Y 474.758,Z 359.081,A -85,B 0,C 180,E1 -7099.336,E2 -7099.336} C_VEL
LIN {X 0,Y 474.362,Z 367.047,A -85,B 0,C 180,E1 -7100.836,E2 -7100.836} C_VEL
LIN {X 0,Y 474.075,Z 373.459,A -85,B 0,C 180,E1 -7102.333,E2 -7102.333} C_VEL
LIN {X 0,Y 473.946,Z 379.144,A -85,B 0,C 180,E1 -7104.042,E2 -7104.042} C_VEL
LIN {X 0,Y 473.759,Z 383.279,A -85,B 0,C 180,E1 -7105.746,E2 -7105.746} C_VEL
LIN {X 0,Y 473.815,Z 384.802,A -85,B 0,C 180,E1 -7106.599,E2 -7106.599} C_VEL
LIN {X 0,Y 473.696,Z 386.828,A -85,B 0,C 180,E1 -7108.3,E2 -7108.3} C_VEL
LIN {X 0,Y 473.668,Z 387.527,A -85,B 0,C 180,E1 -7110,E2 -7110} C_VEL
LIN {X 0,Y 473.695,Z 386.906,A -85,B 0,C 180,E1 -7111.7,E2 -7111.7} C_VEL
LIN {X 0,Y 473.814,Z 384.95,A -85,B 0,C 180,E1 -7113.402,E2 -7113.402} C_VEL
LIN {X 0,Y 473.84,Z 381.617,A -85,B 0,C 180,E1 -7115.106,E2 -7115.106} C_VEL
LIN {X 0,Y 473.981,Z 376.805,A -85,B 0,C 180,E1 -7116.813,E2 -7116.813} C_VEL
LIN {X 0,Y 474.241,Z 370.36,A -85,B 0,C 180,E1 -7118.522,E2 -7118.522} C_VEL
LIN {X 0,Y 474.577,Z 363.183,A -85,B 0,C 180,E1 -7120.021,E2 -7120.021} C_VEL
LIN {X 0,Y 475.002,Z 355.661,A -85,B 0,C 180,E1 -7121.306,E2 -7121.306} C_VEL
LIN {X 0,Y 475.457,Z 345.933,A -85,B 0,C 180,E1 -7122.686,E2 -7122.686} C_VEL
LIN {X 0,Y 476.125,Z 334.643,A -85,B 0,C 180,E1 -7123.988,E2 -7123.988} C_VEL
LIN {X 0,Y 476.749,Z 323.237,A -85,B 0,C 180,E1 -7125.059,E2 -7125.059} C_VEL
LIN {X 0,Y 477.432,Z 310.592,A -85,B 0,C 180,E1 -7126.022,E2 -7126.022} C_VEL
LIN {X 0,Y 477.927,Z 298.543,A -85,B 0,C 180,E1 -7126.76,E2 -7126.76} C_VEL
LIN {X 0,Y 478.457,Z 284.681,A -85,B 0,C 180,E1 -7127.414,E2 -7127.414} C_VEL
LIN {X 0,Y 478.476,Z 277.5,A -85,B 0,C 180,E1 -7127.689,E2 -7127.689} C_VEL
LIN {X 0,Y 475.555,Z 264.569,A -85,B 0,C 180,E1 -7128.179,E2 -7128.179} C_VEL
LIN {X 0,Y 473.961,Z 258.235,A -85,B 0,C 180,E1 -7128.376,E2 -7128.376} C_VEL
LIN {X 0,Y 474.05,Z 252.8,A -85,B 0,C 180,E1 -7131.755,E2 -7131.755} C_VEL
LIN {X 0,Y 474.139,Z 248.424,A -85,B 0,C 180,E1 -7134.522,E2 -7134.522} C_VEL
LIN {X 0,Y 474.21,Z 244.127,A -85,B 0,C 180,E1 -7137.351,E2 -7137.351} C_VEL
LIN {X 0,Y 474.416,Z 239.064,A -85,B 0,C 180,E1 -7140.771,E2 -7140.771} C_VEL
LIN {X 0,Y 474.588,Z 234.067,A -85,B 0,C 180,E1 -7144.245,E2 -7144.245} C_VEL
LIN {X 0,Y 474.631,Z 229.721,A -85,B 0,C 180,E1 -7147.38,E2 -7147.38} C_VEL
LIN {X 0,Y 474.589,Z 226.999,A -85,B 0,C 180,E1 -7149.552,E2 -7149.552} C_VEL
LIN {X 0,Y 474.625,Z 226.989,A -85,B 0,C 180,E1 -7152.236,E2 -7152.236} C_VEL
LIN {X 0,Y 474.623,Z 226.989,A -85,B 0,C 180,E1 -7155.297,E2 -7155.297} C_VEL
LIN {X 0,Y 474.607,Z 226.993,A -85,B 0,C 180,E1 -7158.213,E2 -7158.213} C_VEL
LIN {X 0,Y 474.612,Z 226.991,A -85,B 0,C 180,E1 -7161.543,E2 -7161.543} C_VEL
LIN {X 0,Y 474.626,Z 226.989,A -85,B 0,C 180,E1 -7164.726,E2 -7164.726} C_VEL
LIN {X 0,Y 474.637,Z 226.99,A -85,B 0,C 180,E1 -7167.788,E2 -7167.788} C_VEL
LIN {X 0,Y 474.624,Z 226.992,A -85,B 0,C 180,E1 -7170.885,E2 -7170.885} C_VEL
LIN {X 0,Y 474.657,Z 226.984,A -85,B 0,C 180,E1 -7173.628,E2 -7173.628} C_VEL
LIN {X 0,Y 474.638,Z 226.986,A -85,B 0,C 180,E1 -7176.642,E2 -7176.642} C_VEL
LIN {X 0,Y 474.656,Z 226.983,A -85,B 0,C 180,E1 -7180.09,E2 -7180.09} C_VEL
LIN {X 0,Y 474.639,Z 226.986,A -85,B 0,C 180,E1 -7182.774,E2 -7182.774} C_VEL
LIN {X 0,Y 474.649,Z 226.989,A -85,B 0,C 180,E1 -7185.421,E2 -7185.421} C_VEL
LIN {X 0,Y 474.708,Z 226.977,A -85,B 0,C 180,E1 -7188.038,E2 -7188.038} C_VEL
LIN {X 0,Y 474.714,Z 226.977,A -85,B 0,C 180,E1 -7191.486,E2 -7191.486} C_VEL
LIN {X 0,Y 474.774,Z 226.969,A -85,B 0,C 180,E1 -7194.052,E2 -7194.052} C_VEL
LIN {X 0,Y 474.886,Z 226.954,A -85,B 0,C 180,E1 -7197.455,E2 -7197.455} C_VEL
LIN {X 0,Y 474.841,Z 226.96,A -85,B 0,C 180,E1 -7200.848,E2 -7200.848} C_VEL
LIN {X 0,Y 474.897,Z 226.952,A -85,B 0,C 180,E1 -7202.545,E2 -7202.545} C_VEL
LIN {X 0,Y 474.752,Z 226.972,A -85,B 0,C 180,E1 -7205.948,E2 -7205.948} C_VEL
LIN {X 0,Y 474.699,Z 226.98,A -85,B 0,C 180,E1 -7208.514,E2 -7208.514} C_VEL
LIN {X 0,Y 474.708,Z 226.977,A -85,B 0,C 180,E1 -7211.962,E2 -7211.962} C_VEL
LIN {X 0,Y 474.703,Z 226.978,A -85,B 0,C 180,E1 -7215.456,E2 -7215.456} C_VEL
LIN {X 0,Y 474.663,Z 226.983,A -85,B 0,C 180,E1 -7219.01,E2 -7219.01} C_VEL
LIN {X 0,Y 474.592,Z 226.992,A -85,B 0,C 180,E1 -7221.729,E2 -7221.729} C_VEL
LIN {X 0,Y 474.633,Z 226.989,A -85,B 0,C 180,E1 -7224.494,E2 -7224.494} C_VEL
LIN {X 0,Y 474.604,Z 226.992,A -85,B 0,C 180,E1 -7227.326,E2 -7227.326} C_VEL
LIN {X 0,Y 474.6,Z 226.991,A -85,B 0,C 180,E1 -7230.231,E2 -7230.231} C_VEL
LIN {X 0,Y 474.645,Z 226.985,A -85,B 0,C 180,E1 -7233.22,E2 -7233.22} C_VEL
LIN {X 0,Y 474.586,Z 226.995,A -85,B 0,C 180,E1 -7236.324,E2 -7236.324} C_VEL
LIN {X 0,Y 474.62,Z 226.989,A -85,B 0,C 180,E1 -7239.646,E2 -7239.646} C_VEL
LIN {X 0,Y 474.616,Z 226.993,A -85,B 0,C 180,E1 -7242.934,E2 -7242.934} C_VEL
LIN {X 0,Y 474.604,Z 226.994,A -85,B 0,C 180,E1 -7245.894,E2 -7245.894} C_VEL
LIN {X 0,Y 474.634,Z 227.069,A -85,B 0,C 180,E1 -7248.216,E2 -7248.216} C_VEL
LIN {X 0,Y 475.232,Z 231.011,A -85,B 0,C 180,E1 -7250.512,E2 -7250.512} C_VEL
LIN {X 0,Y 475.324,Z 234.947,A -85,B 0,C 180,E1 -7252.683,E2 -7252.683} C_VEL
LIN {X 0,Y 475.075,Z 241.159,A -85,B 0,C 180,E1 -7255.938,E2 -7255.938} C_VEL
LIN {X 0,Y 474.873,Z 247.527,A -85,B 0,C 180,E1 -7259.136,E2 -7259.136} C_VEL
LIN {X 0,Y 474.679,Z 253.84,A -85,B 0,C 180,E1 -7262.2,E2 -7262.2} C_VEL
LIN {X 0,Y 474.355,Z 260.835,A -85,B 0,C 180,E1 -7265.49,E2 -7265.49} C_VEL
LIN {X 0,Y 474.191,Z 266.761,A -85,B 0,C 180,E1 -7268.252,E2 -7268.252} C_VEL
LIN {X 0,Y 474.042,Z 272.685,A -85,B 0,C 180,E1 -7270.964,E2 -7270.964} C_VEL
LIN {X 0,Y 474.015,Z 274.429,A -85,B 0,C 180,E1 -7271.658,E2 -7271.658} C_VEL
LIN {X 0,Y 477.138,Z 289.244,A -85,B 0,C 180,E1 -7272.127,E2 -7272.127} C_VEL
LIN {X 0,Y 478.465,Z 297.356,A -85,B 0,C 180,E1 -7272.448,E2 -7272.448} C_VEL
LIN {X 0,Y 478.027,Z 311,A -85,B 0,C 180,E1 -7273.027,E2 -7273.027} C_VEL
LIN {X 0,Y 477.354,Z 324.117,A -85,B 0,C 180,E1 -7273.756,E2 -7273.756} C_VEL
LIN {X 0,Y 476.741,Z 336.261,A -85,B 0,C 180,E1 -7274.612,E2 -7274.612} C_VEL
LIN {X 0,Y 476.101,Z 348.517,A -85,B 0,C 180,E1 -7275.685,E2 -7275.685} C_VEL
LIN {X 0,Y 475.51,Z 358.631,A -85,B 0,C 180,E1 -7276.756,E2 -7276.756} C_VEL
LIN {X 0,Y 475.025,Z 368.688,A -85,B 0,C 180,E1 -7278.046,E2 -7278.046} C_VEL
LIN {X 0,Y 474.588,Z 377.041,A -85,B 0,C 180,E1 -7279.332,E2 -7279.332} C_VEL
LIN {X 0,Y 474.221,Z 385.028,A -85,B 0,C 180,E1 -7280.833,E2 -7280.833} C_VEL
LIN {X 0,Y 473.972,Z 391.459,A -85,B 0,C 180,E1 -7282.331,E2 -7282.331} C_VEL
LIN {X 0,Y 473.835,Z 397.162,A -85,B 0,C 180,E1 -7284.04,E2 -7284.04} C_VEL
LIN {X 0,Y 473.821,Z 399.417,A -85,B 0,C 180,E1 -7284.894,E2 -7284.894} C_VEL
LIN {X 0,Y 473.755,Z 402.824,A -85,B 0,C 180,E1 -7286.598,E2 -7286.598} C_VEL
LIN {X 0,Y 473.692,Z 404.839,A -85,B 0,C 180,E1 -7288.3,E2 -7288.3} C_VEL
LIN {X 0,Y 473.667,Z 405.507,A -85,B 0,C 180,E1 -7290,E2 -7290} C_VEL
LIN {X 0,Y 473.692,Z 404.841,A -85,B 0,C 180,E1 -7291.7,E2 -7291.7} C_VEL
LIN {X 0,Y 473.755,Z 402.828,A -85,B 0,C 180,E1 -7293.402,E2 -7293.402} C_VEL
LIN {X 0,Y 473.821,Z 399.421,A -85,B 0,C 180,E1 -7295.106,E2 -7295.106} C_VEL
LIN {X 0,Y 473.892,Z 394.515,A -85,B 0,C 180,E1 -7296.814,E2 -7296.814} C_VEL
LIN {X 0,Y 474.094,Z 387.969,A -85,B 0,C 180,E1 -7298.525,E2 -7298.525} C_VEL
LIN {X 0,Y 474.392,Z 380.685,A -85,B 0,C 180,E1 -7300.025,E2 -7300.025} C_VEL
LIN {X 0,Y 474.908,Z 371.668,A -85,B 0,C 180,E1 -7301.524,E2 -7301.524} C_VEL
LIN {X 0,Y 475.38,Z 362.204,A -85,B 0,C 180,E1 -7302.812,E2 -7302.812} C_VEL
LIN {X 0,Y 475.921,Z 351.728,A -85,B 0,C 180,E1 -7303.993,E2 -7303.993} C_VEL
LIN {X 0,Y 476.508,Z 340.171,A -85,B 0,C 180,E1 -7305.067,E2 -7305.067} C_VEL
LIN {X 0,Y 477.195,Z 327.352,A -85,B 0,C 180,E1 -7306.03,E2 -7306.03} C_VEL
LIN {X 0,Y 477.891,Z 314.087,A -85,B 0,C 180,E1 -7306.816,E2 -7306.816} C_VEL
LIN {X 0,Y 478.346,Z 300.915,A -85,B 0,C 180,E1 -7307.418,E2 -7307.418} C_VEL
LIN {X 0,Y 478.316,Z 295.409,A -85,B 0,C 180,E1 -7307.627,E2 -7307.627} C_VEL
LIN {X 0,Y 475.49,Z 281.195,A -85,B 0,C 180,E1 -7308.148,E2 -7308.148} C_VEL
LIN {X 0,Y 474.015,Z 274.18,A -85,B 0,C 180,E1 -7308.359,E2 -7308.359} C_VEL
LIN {X 0,Y 474.197,Z 268.421,A -85,B 0,C 180,E1 -7310.979,E2 -7310.979} C_VEL
LIN {X 0,Y 474.314,Z 262.802,A -85,B 0,C 180,E1 -7313.582,E2 -7313.582} C_VEL
LIN {X 0,Y 474.594,Z 255.832,A -85,B 0,C 180,E1 -7316.85,E2 -7316.85} C_VEL
LIN {X 0,Y 474.743,Z 250.825,A -85,B 0,C 180,E1 -7319.244,E2 -7319.244} C_VEL
LIN {X 0,Y 474.943,Z 244.838,A -85,B 0,C 180,E1 -7322.189,E2 -7322.189} C_VEL
LIN {X 0,Y 475.202,Z 238.231,A -85,B 0,C 180,E1 -7325.568,E2 -7325.568} C_VEL
LIN {X 0,Y 475.341,Z 232.915,A -85,B 0,C 180,E1 -7328.407,E2 -7328.407} C_VEL
LIN {X 0,Y 474.895,Z 228.368,A -85,B 0,C 180,E1 -7330.996,E2 -7330.996} C_VEL
LIN {X 0,Y 474.612,Z 226.993,A -85,B 0,C 180,E1 -7331.898,E2 -7331.898} C_VEL
LIN {X 0,Y 474.617,Z 226.993,A -85,B 0,C 180,E1 -7335.298,E2 -7335.298} C_VEL
LIN {X 0,Y 474.622,Z 226.99,A -85,B 0,C 180,E1 -7338.215,E2 -7338.215} C_VEL
LIN {X 0,Y 474.611,Z 226.992,A -85,B 0,C 180,E1 -7341.543,E2 -7341.543} C_VEL
LIN {X 0,Y 474.623,Z 226.991,A -85,B 0,C 180,E1 -7344.725,E2 -7344.725} C_VEL
LIN {X 0,Y 474.637,Z 226.99,A -85,B 0,C 180,E1 -7347.788,E2 -7347.788} C_VEL
LIN {X 0,Y 474.602,Z 226.995,A -85,B 0,C 180,E1 -7350.89,E2 -7350.89} C_VEL
LIN {X 0,Y 474.604,Z 226.991,A -85,B 0,C 180,E1 -7353.625,E2 -7353.625} C_VEL
LIN {X 0,Y 474.636,Z 226.986,A -85,B 0,C 180,E1 -7356.642,E2 -7356.642} C_VEL
LIN {X 0,Y 474.653,Z 226.985,A -85,B 0,C 180,E1 -7360.09,E2 -7360.09} C_VEL
LIN {X 0,Y 474.629,Z 226.986,A -85,B 0,C 180,E1 -7362.774,E2 -7362.774} C_VEL
LIN {X 0,Y 474.654,Z 226.986,A -85,B 0,C 180,E1 -7365.421,E2 -7365.421} C_VEL
LIN {X 0,Y 474.707,Z 226.977,A -85,B 0,C 180,E1 -7368.038,E2 -7368.038} C_VEL
LIN {X 0,Y 474.698,Z 226.979,A -85,B 0,C 180,E1 -7371.486,E2 -7371.486} C_VEL
LIN {X 0,Y 474.75,Z 226.972,A -85,B 0,C 180,E1 -7374.052,E2 -7374.052} C_VEL
LIN {X 0,Y 474.896,Z 226.953,A -85,B 0,C 180,E1 -7377.455,E2 -7377.455} C_VEL
LIN {X 0,Y 474.91,Z 226.956,A -85,B 0,C 180,E1 -7380,E2 -7380} C_VEL
LIN {X 0,Y 474.884,Z 226.955,A -85,B 0,C 180,E1 -7382.545,E2 -7382.545} C_VEL
LIN {X 0,Y 474.772,Z 226.969,A -85,B 0,C 180,E1 -7385.948,E2 -7385.948} C_VEL
LIN {X 0,Y 474.729,Z 226.975,A -85,B 0,C 180,E1 -7388.514,E2 -7388.514} C_VEL
LIN {X 0,Y 474.707,Z 226.977,A -85,B 0,C 180,E1 -7391.962,E2 -7391.962} C_VEL
LIN {X 0,Y 474.702,Z 226.977,A -85,B 0,C 180,E1 -7395.456,E2 -7395.456} C_VEL
LIN {X 0,Y 474.667,Z 226.983,A -85,B 0,C 180,E1 -7399.01,E2 -7399.01} C_VEL
LIN {X 0,Y 474.59,Z 226.991,A -85,B 0,C 180,E1 -7401.729,E2 -7401.729} C_VEL
LIN {X 0,Y 474.642,Z 226.988,A -85,B 0,C 180,E1 -7404.494,E2 -7404.494} C_VEL
LIN {X 0,Y 474.682,Z 226.983,A -85,B 0,C 180,E1 -7407.334,E2 -7407.334} C_VEL
LIN {X 0,Y 474.605,Z 226.994,A -85,B 0,C 180,E1 -7410.81,E2 -7410.81} C_VEL
LIN {X 0,Y 474.627,Z 226.987,A -85,B 0,C 180,E1 -7413.221,E2 -7413.221} C_VEL
LIN {X 0,Y 474.59,Z 226.992,A -85,B 0,C 180,E1 -7416.324,E2 -7416.324} C_VEL
LIN {X 0,Y 474.623,Z 226.987,A -85,B 0,C 180,E1 -7419.548,E2 -7419.548} C_VEL
LIN {X 0,Y 474.591,Z 226.997,A -85,B 0,C 180,E1 -7422.232,E2 -7422.232} C_VEL
LIN {X 0,Y 474.618,Z 226.993,A -85,B 0,C 180,E1 -7425.298,E2 -7425.298} C_VEL
LIN {X 0,Y 474.616,Z 226.992,A -85,B 0,C 180,E1 -7428.214,E2 -7428.214} C_VEL
LIN {X 0,Y 474.618,Z 226.993,A -85,B 0,C 180,E1 -7430.451,E2 -7430.451} C_VEL
LIN {X 0,Y 474.647,Z 229.585,A -85,B 0,C 180,E1 -7432.621,E2 -7432.621} C_VEL
LIN {X 0,Y 474.588,Z 233.93,A -85,B 0,C 180,E1 -7435.755,E2 -7435.755} C_VEL
LIN {X 0,Y 474.414,Z 238.918,A -85,B 0,C 180,E1 -7439.229,E2 -7439.229} C_VEL
LIN {X 0,Y 474.208,Z 244.177,A -85,B 0,C 180,E1 -7442.777,E2 -7442.777} C_VEL
LIN {X 0,Y 474.138,Z 248.28,A -85,B 0,C 180,E1 -7445.478,E2 -7445.478} C_VEL
LIN {X 0,Y 474.049,Z 252.655,A -85,B 0,C 180,E1 -7448.245,E2 -7448.245} C_VEL
LIN {X 0,Y 473.968,Z 257.499,A -85,B 0,C 180,E1 -7451.262,E2 -7451.262} C_VEL
LIN {X 0,Y 474.027,Z 258.844,A -85,B 0,C 180,E1 -7451.542,E2 -7451.542} C_VEL
LIN {X 0,Y 474.135,Z 262.027,A -85,B 0,C 180,E1 -7451.778,E2 -7451.778} C_VEL
LIN {X 0,Y 473.701,Z 271.328,A -85,B 0,C 180,E1 -7452.017,E2 -7452.017} C_VEL
LIN {X 0,Y 471.834,Z 285.192,A -85,B 0,C 180,E1 -7452.436,E2 -7452.436} C_VEL
LIN {X 0,Y 471.651,Z 287.48,A -85,B 0,C 180,E1 -7452.533,E2 -7452.533} C_VEL
LIN {X 0,Y 471.063,Z 300.896,A -85,B 0,C 180,E1 -7453.205,E2 -7453.205} C_VEL
LIN {X 0,Y 470.421,Z 314.098,A -85,B 0,C 180,E1 -7454.067,E2 -7454.067} C_VEL
LIN {X 0,Y 469.758,Z 326.055,A -85,B 0,C 180,E1 -7455.044,E2 -7455.044} C_VEL
LIN {X 0,Y 469.061,Z 336.959,A -85,B 0,C 180,E1 -7456.129,E2 -7456.129} C_VEL
LIN {X 0,Y 468.366,Z 347.551,A -85,B 0,C 180,E1 -7457.411,E2 -7457.411} C_VEL
LIN {X 0,Y 467.936,Z 356.585,A -85,B 0,C 180,E1 -7458.741,E2 -7458.741} C_VEL
LIN {X 0,Y 467.446,Z 365.079,A -85,B 0,C 180,E1 -7460.262,E2 -7460.262} C_VEL
LIN {X 0,Y 467.127,Z 371.919,A -85,B 0,C 180,E1 -7461.783,E2 -7461.783} C_VEL
LIN {X 0,Y 466.89,Z 377.861,A -85,B 0,C 180,E1 -7463.458,E2 -7463.458} C_VEL
LIN {X 0,Y 466.784,Z 381.532,A -85,B 0,C 180,E1 -7464.817,E2 -7464.817} C_VEL
LIN {X 0,Y 466.725,Z 384.938,A -85,B 0,C 180,E1 -7466.547,E2 -7466.547} C_VEL
LIN {X 0,Y 466.606,Z 386.964,A -85,B 0,C 180,E1 -7468.274,E2 -7468.274} C_VEL
LIN {X 0,Y 466.597,Z 387.661,A -85,B 0,C 180,E1 -7470,E2 -7470} C_VEL
LIN {X 0,Y 466.605,Z 387.04,A -85,B 0,C 180,E1 -7471.726,E2 -7471.726} C_VEL
LIN {X 0,Y 466.724,Z 385.084,A -85,B 0,C 180,E1 -7473.453,E2 -7473.453} C_VEL
LIN {X 0,Y 466.781,Z 381.75,A -85,B 0,C 180,E1 -7475.183,E2 -7475.183} C_VEL
LIN {X 0,Y 466.913,Z 376.938,A -85,B 0,C 180,E1 -7476.916,E2 -7476.916} C_VEL
LIN {X 0,Y 467.184,Z 370.494,A -85,B 0,C 180,E1 -7478.652,E2 -7478.652} C_VEL
LIN {X 0,Y 467.527,Z 363.317,A -85,B 0,C 180,E1 -7480.174,E2 -7480.174} C_VEL
LIN {X 0,Y 468.028,Z 355.793,A -85,B 0,C 180,E1 -7481.477,E2 -7481.477} C_VEL
LIN {X 0,Y 468.476,Z 346.594,A -85,B 0,C 180,E1 -7482.807,E2 -7482.807} C_VEL
LIN {X 0,Y 469.155,Z 335.814,A -85,B 0,C 180,E1 -7484.089,E2 -7484.089} C_VEL
LIN {X 0,Y 469.801,Z 324.652,A -85,B 0,C 180,E1 -7485.177,E2 -7485.177} C_VEL
LIN {X 0,Y 470.542,Z 312.298,A -85,B 0,C 180,E1 -7486.152,E2 -7486.152} C_VEL
LIN {X 0,Y 471.113,Z 299.258,A -85,B 0,C 180,E1 -7486.977,E2 -7486.977} C_VEL
LIN {X 0,Y 471.68,Z 284.804,A -85,B 0,C 180,E1 -7487.673,E2 -7487.673} C_VEL
LIN {X 0,Y 471.675,Z 278.552,A -85,B 0,C 180,E1 -7487.918,E2 -7487.918} C_VEL
LIN {X 0,Y 468.612,Z 264.969,A -85,B 0,C 180,E1 -7488.451,E2 -7488.451} C_VEL
LIN {X 0,Y 466.898,Z 258.341,A -85,B 0,C 180,E1 -7488.678,E2 -7488.678} C_VEL
LIN {X 0,Y 466.98,Z 254.371,A -85,B 0,C 180,E1 -7491.174,E2 -7491.174} C_VEL
LIN {X 0,Y 467.063,Z 249.993,A -85,B 0,C 180,E1 -7493.971,E2 -7493.971} C_VEL
LIN {X 0,Y 467.114,Z 245.66,A -85,B 0,C 180,E1 -7496.832,E2 -7496.832} C_VEL
LIN {X 0,Y 467.268,Z 241.358,A -85,B 0,C 180,E1 -7499.758,E2 -7499.758} C_VEL
LIN {X 0,Y 467.411,Z 237.22,A -85,B 0,C 180,E1 -7502.646,E2 -7502.646} C_VEL
LIN {X 0,Y 467.552,Z 234.143,A -85,B 0,C 180,E1 -7504.834,E2 -7504.834} C_VEL
LIN {X 0,Y 467.602,Z 229.797,A -85,B 0,C 180,E1 -7508.041,E2 -7508.041} C_VEL
LIN {X 0,Y 467.542,Z 228.337,A -85,B 0,C 180,E1 -7509.149,E2 -7509.149} C_VEL
LIN {X 0,Y 467.553,Z 227.875,A -85,B 0,C 180,E1 -7510.267,E2 -7510.267} C_VEL
LIN {X 0,Y 467.589,Z 227.866,A -85,B 0,C 180,E1 -7512.567,E2 -7512.567} C_VEL
LIN {X 0,Y 467.573,Z 227.869,A -85,B 0,C 180,E1 -7515.053,E2 -7515.053} C_VEL
LIN {X 0,Y 467.568,Z 227.867,A -85,B 0,C 180,E1 -7518.725,E2 -7518.725} C_VEL
LIN {X 0,Y 467.566,Z 227.867,A -85,B 0,C 180,E1 -7521.955,E2 -7521.955} C_VEL
LIN {X 0,Y 467.561,Z 227.867,A -85,B 0,C 180,E1 -7525.167,E2 -7525.167} C_VEL
LIN {X 0,Y 467.584,Z 227.865,A -85,B 0,C 180,E1 -7528.26,E2 -7528.26} C_VEL
LIN {X 0,Y 467.577,Z 227.867,A -85,B 0,C 180,E1 -7531.25,E2 -7531.25} C_VEL
LIN {X 0,Y 467.6,Z 227.865,A -85,B 0,C 180,E1 -7534.159,E2 -7534.159} C_VEL
LIN {X 0,Y 467.579,Z 227.867,A -85,B 0,C 180,E1 -7536.996,E2 -7536.996} C_VEL
LIN {X 0,Y 467.625,Z 227.858,A -85,B 0,C 180,E1 -7539.777,E2 -7539.777} C_VEL
LIN {X 0,Y 467.599,Z 227.865,A -85,B 0,C 180,E1 -7542.506,E2 -7542.506} C_VEL
LIN {X 0,Y 467.608,Z 227.863,A -85,B 0,C 180,E1 -7545.196,E2 -7545.196} C_VEL
LIN {X 0,Y 467.66,Z 227.855,A -85,B 0,C 180,E1 -7547.855,E2 -7547.855} C_VEL
LIN {X 0,Y 467.672,Z 227.853,A -85,B 0,C 180,E1 -7551.357,E2 -7551.357} C_VEL
LIN {X 0,Y 467.738,Z 227.846,A -85,B 0,C 180,E1 -7553.962,E2 -7553.962} C_VEL
LIN {X 0,Y 467.851,Z 227.831,A -85,B 0,C 180,E1 -7557.417,E2 -7557.417} C_VEL
LIN {X 0,Y 467.855,Z 227.834,A -85,B 0,C 180,E1 -7560,E2 -7560} C_VEL
LIN {X 0,Y 467.862,Z 227.828,A -85,B 0,C 180,E1 -7562.583,E2 -7562.583} C_VEL
LIN {X 0,Y 467.715,Z 227.849,A -85,B 0,C 180,E1 -7566.038,E2 -7566.038} C_VEL
LIN {X 0,Y 467.66,Z 227.856,A -85,B 0,C 180,E1 -7568.643,E2 -7568.643} C_VEL
LIN {X 0,Y 467.66,Z 227.854,A -85,B 0,C 180,E1 -7572.145,E2 -7572.145} C_VEL
LIN {X 0,Y 467.642,Z 227.858,A -85,B 0,C 180,E1 -7575.695,E2 -7575.695} C_VEL
LIN {X 0,Y 467.623,Z 227.863,A -85,B 0,C 180,E1 -7579.308,E2 -7579.308} C_VEL
LIN {X 0,Y 467.537,Z 227.87,A -85,B 0,C 180,E1 -7582.074,E2 -7582.074} C_VEL
LIN {X 0,Y 467.572,Z 227.865,A -85,B 0,C 180,E1 -7584.889,E2 -7584.889} C_VEL
LIN {X 0,Y 467.549,Z 227.872,A -85,B 0,C 180,E1 -7587.774,E2 -7587.774} C_VEL
LIN {X 0,Y 467.569,Z 227.869,A -85,B 0,C 180,E1 -7591.044,E2 -7591.044} C_VEL
LIN {X 0,Y 467.59,Z 227.869,A -85,B 0,C 180,E1 -7594.242,E2 -7594.242} C_VEL
LIN {X 0,Y 467.545,Z 227.875,A -85,B 0,C 180,E1 -7597.185,E2 -7597.185} C_VEL
LIN {X 0,Y 467.577,Z 227.869,A -85,B 0,C 180,E1 -7600.265,E2 -7600.265} C_VEL
LIN {X 0,Y 467.589,Z 227.869,A -85,B 0,C 180,E1 -7602.567,E2 -7602.567} C_VEL
LIN {X 0,Y 467.567,Z 227.872,A -85,B 0,C 180,E1 -7605.052,E2 -7605.052} C_VEL
LIN {X 0,Y 467.577,Z 227.997,A -85,B 0,C 180,E1 -7608.02,E2 -7608.02} C_VEL
LIN {X 0,Y 468.094,Z 231.254,A -85,B 0,C 180,E1 -7609.971,E2 -7609.971} C_VEL
LIN {X 0,Y 468.324,Z 234.885,A -85,B 0,C 180,E1 -7612.028,E2 -7612.028} C_VEL
LIN {X 0,Y 468.174,Z 238.83,A -85,B 0,C 180,E1 -7614.165,E2 -7614.165} C_VEL
LIN {X 0,Y 467.953,Z 244.779,A -85,B 0,C 180,E1 -7617.27,E2 -7617.27} C_VEL
LIN {X 0,Y 467.745,Z 250.754,A -85,B 0,C 180,E1 -7620.275,E2 -7620.275} C_VEL
LIN {X 0,Y 467.53,Z 256.747,A -85,B 0,C 180,E1 -7623.194,E2 -7623.194} C_VEL
LIN {X 0,Y 467.233,Z 264.668,A -85,B 0,C 180,E1 -7626.978,E2 -7626.978} C_VEL
LIN {X 0,Y 467.042,Z 270.588,A -85,B 0,C 180,E1 -7629.751,E2 -7629.751} C_VEL
LIN {X 0,Y 466.946,Z 274.17,A -85,B 0,C 180,E1 -7631.368,E2 -7631.368} C_VEL
LIN {X 0,Y 470.096,Z 288.833,A -85,B 0,C 180,E1 -7631.842,E2 -7631.842} C_VEL
LIN {X 0,Y 471.654,Z 298.361,A -85,B 0,C 180,E1 -7632.228,E2 -7632.228} C_VEL
LIN {X 0,Y 471.187,Z 311.93,A -85,B 0,C 180,E1 -7632.825,E2 -7632.825} C_VEL
LIN {X 0,Y 470.417,Z 325.639,A -85,B 0,C 180,E1 -7633.621,E2 -7633.621} C_VEL
LIN {X 0,Y 469.723,Z 338.748,A -85,B 0,C 180,E1 -7634.599,E2 -7634.599} C_VEL
LIN {X 0,Y 469.039,Z 350.527,A -85,B 0,C 180,E1 -7635.686,E2 -7635.686} C_VEL
LIN {X 0,Y 468.466,Z 360.284,A -85,B 0,C 180,E1 -7636.774,E2 -7636.774} C_VEL
LIN {X 0,Y 467.964,Z 370.045,A -85,B 0,C 180,E1 -7638.082,E2 -7638.082} C_VEL
LIN {X 0,Y 467.482,Z 378.142,A -85,B 0,C 180,E1 -7639.388,E2 -7639.388} C_VEL
LIN {X 0,Y 467.13,Z 385.905,A -85,B 0,C 180,E1 -7640.911,E2 -7640.911} C_VEL
LIN {X 0,Y 466.909,Z 391.325,A -85,B 0,C 180,E1 -7642.214,E2 -7642.214} C_VEL
LIN {X 0,Y 466.752,Z 397.027,A -85,B 0,C 180,E1 -7643.95,E2 -7643.95} C_VEL
LIN {X 0,Y 466.635,Z 401.164,A -85,B 0,C 180,E1 -7645.681,E2 -7645.681} C_VEL
LIN {X 0,Y 466.641,Z 403.867,A -85,B 0,C 180,E1 -7647.41,E2 -7647.41} C_VEL
LIN {X 0,Y 466.586,Z 405.206,A -85,B 0,C 180,E1 -7649.137,E2 -7649.137} C_VEL
LIN {X 0,Y 466.586,Z 405.206,A -85,B 0,C 180,E1 -7650.863,E2 -7650.863} C_VEL
LIN {X 0,Y 466.641,Z 403.87,A -85,B 0,C 180,E1 -7652.59,E2 -7652.59} C_VEL
LIN {X 0,Y 466.635,Z 401.168,A -85,B 0,C 180,E1 -7654.319,E2 -7654.319} C_VEL
LIN {X 0,Y 466.754,Z 398.214,A -85,B 0,C 180,E1 -7655.617,E2 -7655.617} C_VEL
LIN {X 0,Y 466.837,Z 392.937,A -85,B 0,C 180,E1 -7657.352,E2 -7657.352} C_VEL
LIN {X 0,Y 467.047,Z 387.833,A -85,B 0,C 180,E1 -7658.655,E2 -7658.655} C_VEL
LIN {X 0,Y 467.352,Z 380.549,A -85,B 0,C 180,E1 -7660.177,E2 -7660.177} C_VEL
LIN {X 0,Y 467.9,Z 371.531,A -85,B 0,C 180,E1 -7661.699,E2 -7661.699} C_VEL
LIN {X 0,Y 468.394,Z 362.066,A -85,B 0,C 180,E1 -7663.007,E2 -7663.007} C_VEL
LIN {X 0,Y 468.997,Z 351.591,A -85,B 0,C 180,E1 -7664.204,E2 -7664.204} C_VEL
LIN {X 0,Y 469.629,Z 340.033,A -85,B 0,C 180,E1 -7665.293,E2 -7665.293} C_VEL
LIN {X 0,Y 470.358,Z 327.213,A -85,B 0,C 180,E1 -7666.27,E2 -7666.27} C_VEL
LIN {X 0,Y 471.059,Z 314.589,A -85,B 0,C 180,E1 -7667.031,E2 -7667.031} C_VEL
LIN {X 0,Y 471.507,Z 302.077,A -85,B 0,C 180,E1 -7667.623,E2 -7667.623} C_VEL
LIN {X 0,Y 471.503,Z 296.414,A -85,B 0,C 180,E1 -7667.848,E2 -7667.848} C_VEL
LIN {X 0,Y 468.672,Z 282.017,A -85,B 0,C 180,E1 -7668.397,E2 -7668.397} C_VEL
LIN {X 0,Y 466.944,Z 274.075,A -85,B 0,C 180,E1 -7668.638,E2 -7668.638} C_VEL
LIN {X 0,Y 467.126,Z 268.604,A -85,B 0,C 180,E1 -7671.167,E2 -7671.167} C_VEL
LIN {X 0,Y 467.269,Z 262.694,A -85,B 0,C 180,E1 -7673.96,E2 -7673.96} C_VEL
LIN {X 0,Y 467.617,Z 255.213,A -85,B 0,C 180,E1 -7677.534,E2 -7677.534} C_VEL
LIN {X 0,Y 467.81,Z 248.739,A -85,B 0,C 180,E1 -7680.716,E2 -7680.716} C_VEL
LIN {X 0,Y 468.023,Z 242.777,A -85,B 0,C 180,E1 -7683.752,E2 -7683.752} C_VEL
LIN {X 0,Y 468.293,Z 236.835,A -85,B 0,C 180,E1 -7686.892,E2 -7686.892} C_VEL
